	out_flg_busy : BOOL;
	out_flg_Done : BOOL;
	out_var_X : LREAL;
	out_var_Y : LREAL;
	out_var_Z : LREAL;
END_VAR
VAR
	fbi_r_TRIG: R_TRIG;
	var_buf_cavNo: INT;
	var_buf_pocketNo: INT;
	var_xLineNo: INT;
	var_yColmnNo: INT;
	var_foo: INT;
	var_vecP12: LREAL;
	var_vecP13: LREAL;
	var_pitchP13: LREAL;
	var_pitchP12: LREAL;
	var_targetPosX: LREAL;
	var_targetPosY: LREAL;
	var_matrix : ARRAY [1..3, 1..3] OF LREAL;
	var_a: LREAL;
	var_b: LREAL;
	var_c: LREAL;
	var_d: LREAL;
	var_buf_calMode: eP_calculateMode;
	//homography
	var_matrixHomo: ARRAY[0..7] OF ARRAY[0..7] OF LREAL;
	var_originPosX: ARRAY[0..3] OF LREAL;
	var_originPosY: ARRAY[0..3] OF LREAL;
	var_marixPivot: ARRAY[0..7] OF LREAL;
	var_i: INT;
	var_j: INT;
	var_pivot: INT;
	//var_matrixA: ARRAY[0..7] OF ARRAY [0..7] OF LREAL;
	//var_amax: LREAL;
	//var_Tmp: LREAL;
	//var_aryPivot: ARRAY[0..7] OF LREAL;
	//var_j: INT;
	
	var_matrixC: ARRAY[0..7] OF ARRAY[0..7] OF LREAL;
	var_matrixD: ARRAY[0..7] OF ARRAY[0..7] OF LREAL;
	var_hi: INT;
	var_aryA: ARRAY[0..7] OF  LREAL;
	
	
END_VAR

fbi_r_TRIG(CLK:= in_flg_run, Q=> );
out_flg_run := in_flg_run;

IF fbi_r_TRIG.Q THEN
	var_buf_cavNo := in_var_cavNo;
	var_buf_pocketNo := in_var_pocketNo;
	var_buf_calMode := in_var_calculateMode;
	out_flg_busy := TRUE;
END_IF

IF out_flg_Done THEN
	out_flg_busy := FALSE;
END_IF
//caluculate target pocket no
IF out_flg_busy THEN
		IF var_ref_productInfo.bottomPocketQty <> 0 THEN
			var_foo := DINT_TO_INT(TRUNC(var_buf_pocketNo / var_ref_productInfo.bottomPocketQty));
		END_IF
	IF var_foo < 1 THEN
		var_xLineNo := var_buf_pocketNo;
		var_yColmnNo := 1;
	ELSIF var_foo >= 1 THEN
		IF var_foo * var_ref_productInfo.bottomPocketQty = in_var_pocketNo THEN
			var_xLineNo := var_buf_pocketNo - (var_ref_productInfo.bottomPocketQty * (var_foo-1));
			var_yColmnNo := var_foo ;
		ELSE
			var_xLineNo := var_buf_pocketNo - (var_ref_productInfo.bottomPocketQty * var_foo);
			var_yColmnNo := var_foo + 1;
		END_IF
	END_IF

    (*          
    
                      back         
      X - - P[2] ---------------- P[1] 
           /                    /|
          /        tray        / |
         /                    /  Z
        /                    /
       P[4]------------------ P[3]
                           /
                          /
                         Y
	          front
	*)
	

//-----------------------------------------------------------------------------------------------------------------------------
	CASE var_buf_calMode OF
		eP_calculateMode.Affine:
			//length
			var_vecP12 := SQRT(EXPT((var_ref_productInfo.teachPos.palletize.upperLower[gvl_param.var_currentTrayPos].cav[var_buf_cavNo].Pos[2].x - var_ref_productInfo.teachPos.palletize.upperLower[gvl_param.var_currentTrayPos].cav[var_buf_cavNo].Pos[1].x),2) + EXPT((var_ref_productInfo.teachPos.palletize.upperLower[gvl_param.var_currentTrayPos].cav[var_buf_cavNo].Pos[2].y - var_ref_productInfo.teachPos.palletize.upperLower[gvl_param.var_currentTrayPos].cav[var_buf_cavNo].Pos[1].y),2));
			var_vecP13 := SQRT(EXPT((var_ref_productInfo.teachPos.palletize.upperLower[gvl_param.var_currentTrayPos].cav[var_buf_cavNo].Pos[3].x - var_ref_productInfo.teachPos.palletize.upperLower[gvl_param.var_currentTrayPos].cav[var_buf_cavNo].Pos[1].x),2) + EXPT((var_ref_productInfo.teachPos.palletize.upperLower[gvl_param.var_currentTrayPos].cav[var_buf_cavNo].Pos[3].y - var_ref_productInfo.teachPos.palletize.upperLower[gvl_param.var_currentTrayPos].cav[var_buf_cavNo].Pos[1].y),2));
			
			//pitch
			IF var_ref_productInfo.bottomPocketQty = 1 THEN
				var_pitchP12 := var_vecP12;
				var_pitchP13 := var_vecP13 / (var_ref_productInfo.vertivalPocketQty - 1);
			ELSIF var_ref_productInfo.vertivalPocketQty = 1 THEN
				var_pitchP12 := var_vecP12 / (var_ref_productInfo.bottomPocketQty - 1);
				var_pitchP13 := var_vecP13;
			ELSE
				var_pitchP12 := var_vecP12 / (var_ref_productInfo.bottomPocketQty - 1);
				var_pitchP13 := var_vecP13 / (var_ref_productInfo.vertivalPocketQty - 1);
			END_IF
			
			
			//target coordinate data (origin data)
			var_targetPosX := ((var_xLineNo - 1) * var_pitchP12);
			var_targetPosY := ((var_yColmnNo - 1) * var_pitchP13);
			
			//genarate affine transform matrix
			IF var_vecP12 = 0 THEN
				var_matrix[1,1] := 0;
			 	var_matrix[1,2] := -var_ref_productInfo.teachPos.palletize.upperLower[gvl_param.var_currentTrayPos].cav[var_buf_cavNo].Pos[1].x/var_vecP13+var_ref_productInfo.teachPos.palletize.upperLower[gvl_param.var_currentTrayPos].cav[var_buf_cavNo].Pos[3].x/var_vecP13;
			 	var_matrix[1,3] := var_ref_productInfo.teachPos.palletize.upperLower[gvl_param.var_currentTrayPos].cav[var_buf_cavNo].Pos[1].x;
		
			 	var_matrix[2,1] := 0;
			 	var_matrix[2,2] := -var_ref_productInfo.teachPos.palletize.upperLower[gvl_param.var_currentTrayPos].cav[var_buf_cavNo].Pos[1].y/var_vecP13+var_ref_productInfo.teachPos.palletize.upperLower[gvl_param.var_currentTrayPos].cav[var_buf_cavNo].Pos[3].y/var_vecP13;
			 	var_matrix[2,3] := var_ref_productInfo.teachPos.palletize.upperLower[gvl_param.var_currentTrayPos].cav[var_buf_cavNo].Pos[1].y;
			
			  	var_matrix[3,1] := 0;
			  	var_matrix[3,2] := 0;
			  	var_matrix[3,3] := 1;
			ELSIF var_vecP13 = 0 THEN
				var_matrix[1,1] := -var_ref_productInfo.teachPos.palletize.upperLower[gvl_param.var_currentTrayPos].cav[var_buf_cavNo].Pos[1].x/var_vecP12+var_ref_productInfo.teachPos.palletize.upperLower[gvl_param.var_currentTrayPos].cav[var_buf_cavNo].Pos[2].x/var_vecP12;
			 	var_matrix[1,2] := 0;
			 	var_matrix[1,3] := var_ref_productInfo.teachPos.palletize.upperLower[gvl_param.var_currentTrayPos].cav[var_buf_cavNo].Pos[1].x;
		
			 	var_matrix[2,1] := -var_ref_productInfo.teachPos.palletize.upperLower[gvl_param.var_currentTrayPos].cav[var_buf_cavNo].Pos[1].y/var_vecP12+var_ref_productInfo.teachPos.palletize.upperLower[gvl_param.var_currentTrayPos].cav[var_buf_cavNo].Pos[2].y/var_vecP12;
			 	var_matrix[2,2] := 0;
			 	var_matrix[2,3] := var_ref_productInfo.teachPos.palletize.upperLower[gvl_param.var_currentTrayPos].cav[var_buf_cavNo].Pos[1].y;
			
			  	var_matrix[3,1] := 0;
			  	var_matrix[3,2] := 0;
			  	var_matrix[3,3] := 1;
			ELSE
				var_matrix[1,1] := -var_ref_productInfo.teachPos.palletize.upperLower[gvl_param.var_currentTrayPos].cav[var_buf_cavNo].Pos[1].x/var_vecP12+var_ref_productInfo.teachPos.palletize.upperLower[gvl_param.var_currentTrayPos].cav[var_buf_cavNo].Pos[2].x/var_vecP12;
			 	var_matrix[1,2] := -var_ref_productInfo.teachPos.palletize.upperLower[gvl_param.var_currentTrayPos].cav[var_buf_cavNo].Pos[1].x/var_vecP13+var_ref_productInfo.teachPos.palletize.upperLower[gvl_param.var_currentTrayPos].cav[var_buf_cavNo].Pos[3].x/var_vecP13;
			 	var_matrix[1,3] := var_ref_productInfo.teachPos.palletize.upperLower[gvl_param.var_currentTrayPos].cav[var_buf_cavNo].Pos[1].x;
		
			 	var_matrix[2,1] := -var_ref_productInfo.teachPos.palletize.upperLower[gvl_param.var_currentTrayPos].cav[var_buf_cavNo].Pos[1].y/var_vecP12+var_ref_productInfo.teachPos.palletize.upperLower[gvl_param.var_currentTrayPos].cav[var_buf_cavNo].Pos[2].y/var_vecP12;
			 	var_matrix[2,2] := -var_ref_productInfo.teachPos.palletize.upperLower[gvl_param.var_currentTrayPos].cav[var_buf_cavNo].Pos[1].y/var_vecP13+var_ref_productInfo.teachPos.palletize.upperLower[gvl_param.var_currentTrayPos].cav[var_buf_cavNo].Pos[3].y/var_vecP13;
			 	var_matrix[2,3] := var_ref_productInfo.teachPos.palletize.upperLower[gvl_param.var_currentTrayPos].cav[var_buf_cavNo].Pos[1].y;
			
			  	var_matrix[3,1] := 0;
			  	var_matrix[3,2] := 0;
			  	var_matrix[3,3] := 1;
			END_IF

			  
			  
			  //caluculate Axis Z coordinate data
			var_a := (var_ref_productInfo.teachPos.palletize.upperLower[gvl_param.var_currentTrayPos].cav[var_buf_cavNo].Pos[2].y - var_ref_productInfo.teachPos.palletize.upperLower[gvl_param.var_currentTrayPos].cav[var_buf_cavNo].Pos[1].y) * (var_ref_productInfo.teachPos.palletize.upperLower[gvl_param.var_currentTrayPos].cav[var_buf_cavNo].Pos[3].z - var_ref_productInfo.teachPos.palletize.upperLower[gvl_param.var_currentTrayPos].cav[var_buf_cavNo].Pos[1].z) - (var_ref_productInfo.teachPos.palletize.upperLower[gvl_param.var_currentTrayPos].cav[var_buf_cavNo].Pos[3].y - var_ref_productInfo.teachPos.palletize.upperLower[gvl_param.var_currentTrayPos].cav[var_buf_cavNo].Pos[1].y) * (var_ref_productInfo.teachPos.palletize.upperLower[gvl_param.var_currentTrayPos].cav[var_buf_cavNo].Pos[2].z - var_ref_productInfo.teachPos.palletize.upperLower[gvl_param.var_currentTrayPos].cav[var_buf_cavNo].Pos[1].z);
			var_b := (var_ref_productInfo.teachPos.palletize.upperLower[gvl_param.var_currentTrayPos].cav[var_buf_cavNo].Pos[2].z - var_ref_productInfo.teachPos.palletize.upperLower[gvl_param.var_currentTrayPos].cav[var_buf_cavNo].Pos[1].z) * (var_ref_productInfo.teachPos.palletize.upperLower[gvl_param.var_currentTrayPos].cav[var_buf_cavNo].Pos[3].x - var_ref_productInfo.teachPos.palletize.upperLower[gvl_param.var_currentTrayPos].cav[var_buf_cavNo].Pos[1].x) - (var_ref_productInfo.teachPos.palletize.upperLower[gvl_param.var_currentTrayPos].cav[var_buf_cavNo].Pos[3].z - var_ref_productInfo.teachPos.palletize.upperLower[gvl_param.var_currentTrayPos].cav[var_buf_cavNo].Pos[1].z) * (var_ref_productInfo.teachPos.palletize.upperLower[gvl_param.var_currentTrayPos].cav[var_buf_cavNo].Pos[2].x - var_ref_productInfo.teachPos.palletize.upperLower[gvl_param.var_currentTrayPos].cav[var_buf_cavNo].Pos[1].x);
			var_c := (var_ref_productInfo.teachPos.palletize.upperLower[gvl_param.var_currentTrayPos].cav[var_buf_cavNo].Pos[2].x - var_ref_productInfo.teachPos.palletize.upperLower[gvl_param.var_currentTrayPos].cav[var_buf_cavNo].Pos[1].x) * (var_ref_productInfo.teachPos.palletize.upperLower[gvl_param.var_currentTrayPos].cav[var_buf_cavNo].Pos[3].y - var_ref_productInfo.teachPos.palletize.upperLower[gvl_param.var_currentTrayPos].cav[var_buf_cavNo].Pos[1].y) - (var_ref_productInfo.teachPos.palletize.upperLower[gvl_param.var_currentTrayPos].cav[var_buf_cavNo].Pos[3].x - var_ref_productInfo.teachPos.palletize.upperLower[gvl_param.var_currentTrayPos].cav[var_buf_cavNo].Pos[1].x) * (var_ref_productInfo.teachPos.palletize.upperLower[gvl_param.var_currentTrayPos].cav[var_buf_cavNo].Pos[2].y - var_ref_productInfo.teachPos.palletize.upperLower[gvl_param.var_currentTrayPos].cav[var_buf_cavNo].Pos[1].y);
			var_d := -((var_a * var_ref_productInfo.teachPos.palletize.upperLower[gvl_param.var_currentTrayPos].cav[var_buf_cavNo].Pos[1].x) + (var_b * var_ref_productInfo.teachPos.palletize.upperLower[gvl_param.var_currentTrayPos].cav[var_buf_cavNo].Pos[1].y) + (var_c * var_ref_productInfo.teachPos.palletize.upperLower[gvl_param.var_currentTrayPos].cav[var_buf_cavNo].Pos[1].z));
			
			// caluculate (afiine transform matrix * target coordinate data)
			out_var_X := (var_matrix[1,1] * var_targetPosX) + (var_matrix[1,2] * var_targetPosY) + var_matrix[1,3];
			out_var_Y := (var_matrix[2,1] * var_targetPosX) + (var_matrix[2,2] * var_targetPosY) + var_matrix[2,3];
			IF var_c <> 0 THEN
				out_var_Z := -((var_a * out_var_X) + (var_b * out_var_Y) + var_d) / var_c;
			ELSE
				out_var_Z := var_ref_productInfo.teachPos.palletize.upperLower[gvl_param.var_currentTrayPos].cav[var_buf_cavNo].Pos[1].z;
			END_IF	
			out_flg_Done := TRUE;
		eP_calculateMode.Homography:
			//
			out_flg_Done := FALSE;
	END_CASE

ELSE
	out_flg_Done := FALSE;
	
END_IF

END_FUNCTION_BLOCK

// ---- FBs/fb_operationElecylinder.TcPOU
FUNCTION_BLOCK fb_operationElecylinder
VAR_INPUT
END_VAR
VAR_OUTPUT
END_VAR
VAR
	SFCInit: bool;
	TranPosDone: BOOL;
	TranNegDone: BOOL;
	SamplePosDone: BOOL;
	SampleNegDone: BOOL;
	TrayChangePosDone: BOOL;
	TrayChangeNegDone: BOOL;
	flgInitDone: BOOL;
	trn_RotaryNegDone: BOOL;
	trn_RotaryPosDone: BOOL;
	trn_flgInitDone: BOOL;
	var_process: INT;
END_VAR

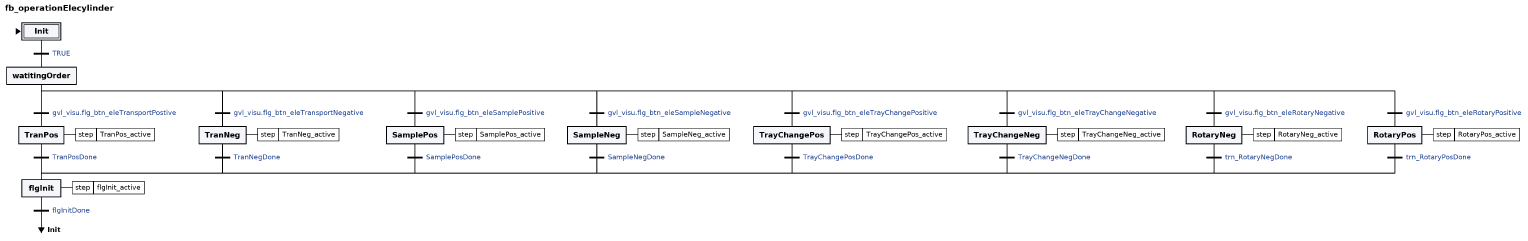
INITIAL_STEP Init:
END_STEP
TRANSITION FROM Init TO watitingOrder
    := TRUE;
END_TRANSITION
STEP watitingOrder:
END_STEP
TRANSITION FROM watitingOrder TO TranPos
    := gvl_visu.flg_btn_eleTransportPostive;
END_TRANSITION
STEP TranPos:
    TranPos_active(N);  // step action
END_STEP
TRANSITION FROM TranPos TO flgInit
    := TranPosDone;
END_TRANSITION
TRANSITION FROM watitingOrder TO TranNeg
    := gvl_visu.flg_btn_eleTransportNegative;
END_TRANSITION
STEP TranNeg:
    TranNeg_active(N);  // step action
END_STEP
TRANSITION FROM TranNeg TO flgInit
    := TranNegDone;
END_TRANSITION
TRANSITION FROM watitingOrder TO SamplePos
    := gvl_visu.flg_btn_eleSamplePositive;
END_TRANSITION
STEP SamplePos:
    SamplePos_active(N);  // step action
END_STEP
TRANSITION FROM SamplePos TO flgInit
    := SamplePosDone;
END_TRANSITION
TRANSITION FROM watitingOrder TO SampleNeg
    := gvl_visu.flg_btn_eleSampleNegative;
END_TRANSITION
STEP SampleNeg:
    SampleNeg_active(N);  // step action
END_STEP
TRANSITION FROM SampleNeg TO flgInit
    := SampleNegDone;
END_TRANSITION
TRANSITION FROM watitingOrder TO TrayChangePos
    := gvl_visu.flg_btn_eleTrayChangePositive;
END_TRANSITION
STEP TrayChangePos:
    TrayChangePos_active(N);  // step action
END_STEP
TRANSITION FROM TrayChangePos TO flgInit
    := TrayChangePosDone;
END_TRANSITION
TRANSITION FROM watitingOrder TO TrayChangeNeg
    := gvl_visu.flg_btn_eleTrayChangeNegative;
END_TRANSITION
STEP TrayChangeNeg:
    TrayChangeNeg_active(N);  // step action
END_STEP
TRANSITION FROM TrayChangeNeg TO flgInit
    := TrayChangeNegDone;
END_TRANSITION
TRANSITION FROM watitingOrder TO RotaryNeg
    := gvl_visu.flg_btn_eleRotaryNegative;
END_TRANSITION
STEP RotaryNeg:
    RotaryNeg_active(N);  // step action
END_STEP
TRANSITION FROM RotaryNeg TO flgInit
    := trn_RotaryNegDone;
END_TRANSITION
TRANSITION FROM watitingOrder TO RotaryPos
    := gvl_visu.flg_btn_eleRotaryPositive;
END_TRANSITION
STEP RotaryPos:
    RotaryPos_active(N);  // step action
END_STEP
TRANSITION FROM RotaryPos TO flgInit
    := trn_RotaryPosDone;
END_TRANSITION
STEP flgInit:
    flgInit_active(N);  // step action
END_STEP
TRANSITION FROM flgInit TO Init
    := flgInitDone;
END_TRANSITION

ACTION flgInit_active:
IF flgInit._x AND flgInit.x = FALSE THEN
	flgInitDone:= FALSE;
	gvl_visu.flg_btn_eleTransportPostive := FALSE;
	gvl_visu.flg_btn_eleTransportNegative := FALSE;
	gvl_visu.flg_btn_eleSamplePositive := FALSE;
	gvl_visu.flg_btn_eleSampleNegative := FALSE;
	gvl_visu.flg_btn_eleTrayChangePositive := FALSE;
	gvl_visu.flg_btn_eleTrayChangeNegative := FALSE;
	gvl_visu.flg_btn_eleRotaryPositive := FALSE;
	gvl_visu.flg_btn_eleRotaryNegative := FALSE;
ELSIF flgInit._x AND flgInit.x THEN
	flgInitDone := TRUE;
END_IF
END_ACTION

PROPERTY p_Init : bool
GET
p_init := THIS^.SFCInit;
END_GET
SET
THIS^.SFCInit := p_init;
END_SET
END_PROPERTY

ACTION RotaryNeg_active:
IF RotaryNeg._x AND RotaryNeg.x = FALSE THEN
	trn_RotaryNegDone := FALSE;
	gvl_elecylinder.fbi_axisRotary.in_flg_run := FALSE;
	gvl_elecylinder.fbi_axisRotary.in_var_moveMode := eP_eleMoveMode.eleA;
	var_process := 0;
ELSIF RotaryNeg._x AND RotaryNeg.x THEN
	CASE var_process OF
		0:
			gvl_elecylinder.fbi_axisRotary.in_flg_run := TRUE;
			var_process := 1;
		1:
			IF gvl_elecylinder.fbi_axisRotary.out_flg_Done THEN
				gvl_elecylinder.fbi_axisRotary.in_flg_run := FALSE;
				trn_RotaryNegDone := TRUE;
			END_IF
	END_CASE
END_IF
END_ACTION

ACTION RotaryPos_active:
IF RotaryPos._x AND RotaryPos.x = FALSE THEN
	trn_RotaryPosDone := FALSE;
	gvl_elecylinder.fbi_axisRotary.in_flg_run := FALSE;
	gvl_elecylinder.fbi_axisRotary.in_var_moveMode := eP_eleMoveMode.eleB;
	var_process := 0;
ELSIF RotaryPos._x AND RotaryPos.x THEN
	CASE var_process OF
		0:
			gvl_elecylinder.fbi_axisRotary.in_flg_run := TRUE;
			var_process :=1;
		1:
			IF gvl_elecylinder.fbi_axisRotary.out_flg_Done THEN
				gvl_elecylinder.fbi_axisRotary.in_flg_run := FALSE;
				trn_RotaryPosDone := TRUE;
			END_IF
	END_CASE
END_IF
END_ACTION

ACTION SampleNeg_active:
IF SampleNeg._x AND SampleNeg.x = FALSE THEN
	SampleNegDone := FALSE;
	gvl_elecylinder.fbi_axisSample.in_flg_run := FALSE;
	gvl_elecylinder.fbi_axisSample.in_var_moveMode := eP_eleMoveMode.eleA;
	var_process := 0;
ELSIF SampleNeg._x AND SampleNeg.x THEN
	CASE var_process OF
		0:
			gvl_elecylinder.fbi_axisSample.in_flg_run := TRUE;
			var_process := 1;
		1:
			IF gvl_elecylinder.fbi_axisSample.out_flg_Done THEN
				gvl_elecylinder.fbi_axisSample.in_flg_run := FALSE;
				SampleNegDone := TRUE;
			END_IF
	END_CASE
END_IF
END_ACTION

ACTION SamplePos_active:
IF SamplePos._x AND SamplePos.x = FALSE THEN
	SamplePosDone := FALSE;
	gvl_elecylinder.fbi_axisSample.in_flg_run := FALSE;
	gvl_elecylinder.fbi_axisSample.in_var_moveMode := eP_eleMoveMode.eleB;
	var_process := 0;
ELSIF SamplePos._x AND SamplePos.x THEN
	CASE var_process OF
		0:
			gvl_elecylinder.fbi_axisSample.in_flg_run := TRUE;
			var_process := 1;
		1:
			IF gvl_elecylinder.fbi_axisSample.out_flg_Done THEN
				gvl_elecylinder.fbi_axisSample.in_flg_run := FALSE;
				SamplePosDone := TRUE;
			END_IF
	END_CASE
END_IF
END_ACTION

ACTION TranNeg_active:
IF TranNeg._x AND TranNeg.x = FALSE THEN
	TranNegDone := FALSE;
	gvl_elecylinder.fbi_axisTransport.in_flg_run := FALSE;
	gvl_elecylinder.fbi_axisTransport.in_var_moveMode := eP_eleMoveMode.eleA;
	var_process := 0;
ELSIF TranNeg._x AND TranNeg.x THEN
	CASE var_process OF
		0:
			gvl_elecylinder.fbi_axisTransport.in_flg_run := TRUE;
			var_process := 1;
		1:
			IF gvl_elecylinder.fbi_axisTransport.out_flg_Done THEN
				gvl_elecylinder.fbi_axisTransport.in_flg_run := FALSE;
				TranNegDone := TRUE;
			END_IF
	END_CASE
END_IF
END_ACTION

ACTION TranPos_active:
IF TranPos._x AND TranPos.x = FALSE THEN
	TranPosDone := FALSE;
	gvl_elecylinder.fbi_axisTransport.in_flg_run := FALSE;
	gvl_elecylinder.fbi_axisTransport.in_var_moveMode := eP_eleMoveMode.eleB;
	var_process := 0;
ELSIF TranPos._x AND TranPos.x THEN
	CASE var_process OF
		0:
			gvl_elecylinder.fbi_axisTransport.in_flg_run := TRUE;
			var_process := 1;
		1:
			IF gvl_elecylinder.fbi_axisTransport.out_flg_Done THEN
				TranPosDone := TRUE;
			END_IF
	END_CASE
END_IF
END_ACTION

ACTION TrayChangeNeg_active:
IF TrayChangeNeg._x AND TrayChangeNeg.x = FALSE THEN
	TrayChangeNegDone := FALSE;
	gvl_elecylinder.fbi_axisTrayChange.in_flg_run := FALSE;
	gvl_elecylinder.fbi_axisTrayChange.in_var_moveMode := eP_eleMoveMode.eleA;
	var_process := 0;
ELSIF TrayChangeNeg._x AND TrayChangeNeg.x THEN
	CASE var_process OF
		0:
			gvl_axis.ref_z.Position := 50;
			gvl_axis.ref_z.Execute := TRUE;
			var_process := 1;
		1:
			IF gvl_axis.ref_z.Done THEN
				gvl_axis.ref_z.Execute := FALSE;
				var_process := 2;
			END_IF
		2:
			gvl_elecylinder.fbi_axisTrayChange.in_flg_run := TRUE;
			var_process := 3;
		3:
			IF gvl_elecylinder.fbi_axisTrayChange.out_flg_Done THEN
				gvl_elecylinder.fbi_axisTrayChange.in_flg_run := FALSE;
				TrayChangeNegDone := TRUE;
			END_IF
	END_CASE
END_IF
END_ACTION

ACTION TrayChangePos_active:
IF TrayChangePos._x AND TrayChangePos.x = FALSE THEN
	TrayChangePosDone := FALSE;
	gvl_elecylinder.fbi_axisTrayChange.in_flg_run := FALSE;
	gvl_elecylinder.fbi_axisTrayChange.in_var_moveMode := eP_eleMoveMode.eleB;
	var_process := 0;
ELSIF TrayChangePos._x AND TrayChangePos.x THEN
	CASE var_process OF
		0:
			gvl_axis.ref_z.Position := 50;
			gvl_axis.ref_z.Execute := TRUE;
			var_process := 1;
		1:
			IF gvl_axis.ref_z.Done THEN
				gvl_axis.ref_z.Execute := FALSE;
				var_process := 2;
			END_IF
		2:
			gvl_elecylinder.fbi_axisTrayChange.in_flg_run := TRUE;
			var_process := 3;
		3:
			IF gvl_elecylinder.fbi_axisTrayChange.out_flg_Done THEN
				gvl_elecylinder.fbi_axisTrayChange.in_flg_run := FALSE;
				TrayChangePosDone := TRUE;
			END_IF
	END_CASE
END_IF
END_ACTION

END_FUNCTION_BLOCK

// ---- FBs/gateMeasurementModule/fb_gm_operationElecylinder.TcPOU
FUNCTION_BLOCK fb_gm_operationElecylinder
VAR_INPUT
END_VAR
VAR_OUTPUT
END_VAR
VAR
	SFCInit: bool;
	TranPosDone: BOOL;
	TranNegDone: BOOL;
	flgInitDone: BOOL;
	PickUpPosDone: BOOL;
	PickUpNegDone: BOOL;
	var_process: INT;
END_VAR

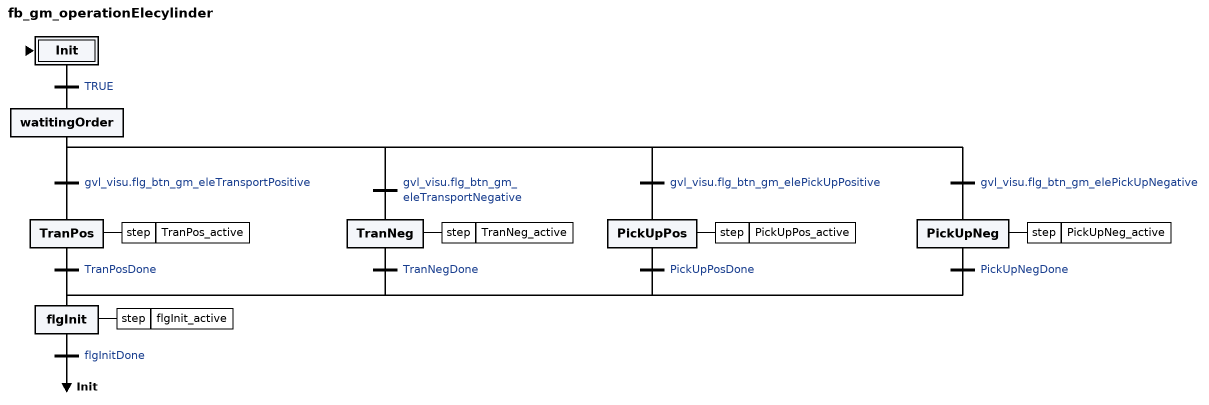
INITIAL_STEP Init:
END_STEP
TRANSITION FROM Init TO watitingOrder
    := TRUE;
END_TRANSITION
STEP watitingOrder:
END_STEP
TRANSITION FROM watitingOrder TO TranPos
    := gvl_visu.flg_btn_gm_eleTransportPositive;
END_TRANSITION
STEP TranPos:
    TranPos_active(N);  // step action
END_STEP
TRANSITION FROM TranPos TO flgInit
    := TranPosDone;
END_TRANSITION
TRANSITION FROM watitingOrder TO TranNeg
    := gvl_visu.flg_btn_gm_eleTransportNegative;
END_TRANSITION
STEP TranNeg:
    TranNeg_active(N);  // step action
END_STEP
TRANSITION FROM TranNeg TO flgInit
    := TranNegDone;
END_TRANSITION
TRANSITION FROM watitingOrder TO PickUpPos
    := gvl_visu.flg_btn_gm_elePickUpPositive;
END_TRANSITION
STEP PickUpPos:
    PickUpPos_active(N);  // step action
END_STEP
TRANSITION FROM PickUpPos TO flgInit
    := PickUpPosDone;
END_TRANSITION
TRANSITION FROM watitingOrder TO PickUpNeg
    := gvl_visu.flg_btn_gm_elePickUpNegative;
END_TRANSITION
STEP PickUpNeg:
    PickUpNeg_active(N);  // step action
END_STEP
TRANSITION FROM PickUpNeg TO flgInit
    := PickUpNegDone;
END_TRANSITION
STEP flgInit:
    flgInit_active(N);  // step action
END_STEP
TRANSITION FROM flgInit TO Init
    := flgInitDone;
END_TRANSITION

ACTION flgInit_active:
IF flgInit._x AND flgInit.x = FALSE THEN
	flgInitDone:= FALSE;
	gvl_visu.flg_btn_gm_eleTransportPositive := FALSE;
	gvl_visu.flg_btn_gm_eleTransportNegative := FALSE;
	gvl_visu.flg_btn_gm_elePickUpPositive := FALSE;
	gvl_visu.flg_btn_gm_elePickUpNegative := FALSE;
	gvl_visu.flg_btn_eleSamplePositive := FALSE;
	gvl_visu.flg_btn_eleSampleNegative := FALSE;
	gvl_visu.flg_btn_eleTrayChangePositive := FALSE;
	gvl_visu.flg_btn_eleTrayChangeNegative := FALSE;
	gvl_visu.flg_btn_eleRotaryPositive := FALSE;
	gvl_visu.flg_btn_eleRotaryNegative := FALSE;
ELSIF flgInit._x AND flgInit.x THEN
	flgInitDone := TRUE;
END_IF
END_ACTION

PROPERTY p_Init : bool
GET
p_init := THIS^.SFCInit;
END_GET
SET
THIS^.SFCInit := p_init;
END_SET
END_PROPERTY

ACTION PickUpNeg_active:
IF PickUpNeg._x AND PickUpNeg.x = FALSE THEN
	PickUpNegDone := FALSE;
	gvl_elecylinder.fbi_gm_axisPickUp.in_flg_run := FALSE;
	gvl_elecylinder.fbi_gm_axisPickUp.in_var_moveMode := eP_eleMoveMode.eleA;
	var_process := 0;
ELSIF PickUpNeg._x AND PickUpNeg.x THEN
	CASE var_process OF
		0:
			gvl_elecylinder.fbi_gm_axisPickUp.in_flg_run := TRUE;
			var_process := 1;
		1:
			IF gvl_elecylinder.fbi_gm_axisPickUp.out_flg_Done THEN
				gvl_elecylinder.fbi_gm_axisPickUp.in_flg_run := FALSE;
				PickUpNegDone := TRUE;
			END_IF
	END_CASE
END_IF
END_ACTION

ACTION PickUpPos_active:
IF PickUpPos._x AND PickUpPos.x = FALSE THEN
	PickUpPosDone := FALSE;
	gvl_elecylinder.fbi_gm_axisPickUp.in_flg_run := FALSE;
	gvl_elecylinder.fbi_gm_axisPickUp.in_var_moveMode := eP_eleMoveMode.eleB;
	var_process := 0;
ELSIF PickUpPos._x AND PickUpPos.x THEN
	CASE var_process OF
		0:
			gvl_elecylinder.fbi_gm_axisPickUp.in_flg_run := TRUE;
			var_process := 1;
		1:
			IF gvl_elecylinder.fbi_gm_axisPickUp.out_flg_Done THEN
				gvl_elecylinder.fbi_gm_axisPickUp.in_flg_run := FALSE;
				PickUpPosDone := TRUE;
			END_IF
	END_CASE
END_IF
END_ACTION

ACTION TranNeg_active:
IF TranNeg._x AND TranNeg.x = FALSE THEN
	TranNegDone := FALSE;
	gvl_elecylinder.fbi_gm_axisTransport.in_flg_run := FALSE;
	gvl_elecylinder.fbi_gm_axisTransport.in_var_moveMode := eP_eleMoveMode.eleA;
	var_process := 0;
ELSIF TranNeg._x AND TranNeg.x THEN
	CASE var_process OF
		0:
			gvl_elecylinder.fbi_gm_axisTransport.in_flg_run := TRUE;
			var_process := 1;
		1:
			IF gvl_elecylinder.fbi_gm_axisTransport.out_flg_Done THEN
				gvl_elecylinder.fbi_gm_axisTransport.in_flg_run := FALSE;
				TranNegDone := TRUE;
			END_IF
	END_CASE
END_IF
END_ACTION

ACTION TranPos_active:
IF TranPos._x AND TranPos.x = FALSE THEN
	TranPosDone := FALSE;
	gvl_elecylinder.fbi_gm_axisTransport.in_flg_run := FALSE;
	gvl_elecylinder.fbi_gm_axisTransport.in_var_moveMode := eP_eleMoveMode.eleB;
	var_process := 0;
ELSIF TranPos._x AND TranPos.x THEN
	CASE var_process OF
		0:
			gvl_elecylinder.fbi_gm_axisTransport.in_flg_run := TRUE;
			var_process := 1;
		1:
			IF gvl_elecylinder.fbi_gm_axisTransport.out_flg_Done THEN
				gvl_elecylinder.fbi_gm_axisTransport.in_flg_run := FALSE;
				TranPosDone := TRUE;
			END_IF
	END_CASE
END_IF
END_ACTION

END_FUNCTION_BLOCK

// ---- FBs/fb_oeprationChuck.TcPOU
FUNCTION_BLOCK fb_oeprationChuck
VAR_INPUT
END_VAR
VAR_OUTPUT
END_VAR
VAR
	SFCInit : bool;
	flgInitDone: BOOL;
	trn_chuckCloseDone: BOOL;
	trn_chuckOpenDone: BOOL;
END_VAR

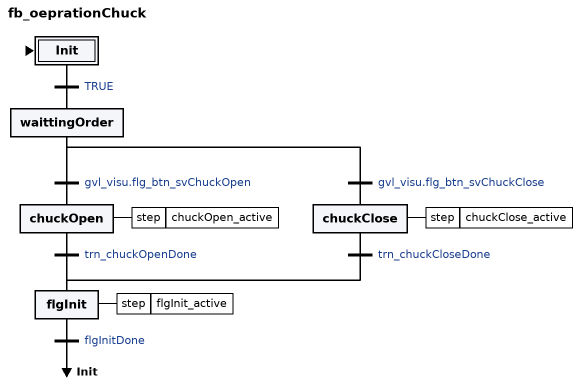
INITIAL_STEP Init:
END_STEP
TRANSITION FROM Init TO waittingOrder
    := TRUE;
END_TRANSITION
STEP waittingOrder:
END_STEP
TRANSITION FROM waittingOrder TO chuckOpen
    := gvl_visu.flg_btn_svChuckOpen;
END_TRANSITION
STEP chuckOpen:
    chuckOpen_active(N);  // step action
END_STEP
TRANSITION FROM chuckOpen TO flgInit
    := trn_chuckOpenDone;
END_TRANSITION
TRANSITION FROM waittingOrder TO chuckClose
    := gvl_visu.flg_btn_svChuckClose;
END_TRANSITION
STEP chuckClose:
    chuckClose_active(N);  // step action
END_STEP
TRANSITION FROM chuckClose TO flgInit
    := trn_chuckCloseDone;
END_TRANSITION
STEP flgInit:
    flgInit_active(N);  // step action
END_STEP
TRANSITION FROM flgInit TO Init
    := flgInitDone;
END_TRANSITION

ACTION chuckClose_active:
IF chuckClose._x AND chuckClose.x = FALSE THEN
	trn_chuckCloseDone := FALSE;
	gvl_solv.fbi_chuck.in_flg_run := FALSE;
	gvl_solv.fbi_chuck.in_var_moveMode := eP_svMoveMode.svB;
ELSIF chuckClose._x AND chuckClose.x THEN
	gvl_solv.fbi_chuck.in_flg_run := TRUE;
	IF gvl_solv.fbi_chuck.out_flg_Done THEN
		gvl_solv.fbi_chuck.in_flg_run := FALSE;
		trn_chuckCloseDone := TRUE;
	END_IF
END_IF
END_ACTION

ACTION chuckOpen_active:
IF chuckOpen._x AND chuckOpen.x = FALSE THEN
	trn_chuckOpenDone := FALSE;
	gvl_solv.fbi_chuck.in_flg_run := FALSE;
	gvl_solv.fbi_chuck.in_var_moveMode := eP_svMoveMode.svA;
ELSIF chuckOpen._x AND chuckOpen.x THEN
	gvl_solv.fbi_chuck.in_flg_run := TRUE;
	IF gvl_solv.fbi_chuck.out_flg_Done THEN
		gvl_solv.fbi_chuck.in_flg_run := FALSE;
		trn_chuckOpenDone := TRUE;
	END_IF
END_IF
END_ACTION

ACTION flgInit_active:
IF flgInit._x AND flgInit.x = FALSE THEN
	flgInitDone := FALSE;
	gvl_visu.flg_btn_svChuckOpen := FALSE;
	gvl_visu.flg_btn_svChuckClose := FALSE;
ELSIF flgInit._x AND flgInit.x THEN
	flgInitDone := TRUE;
END_IF
END_ACTION

PROPERTY p_Init : bool
GET
p_init := THIS^.SFCInit;
END_GET
SET
THIS^.SFCInit := p_Init;
END_SET
END_PROPERTY

END_FUNCTION_BLOCK

// ---- FBs/fb_oeprationPush.TcPOU
FUNCTION_BLOCK fb_oeprationPush
VAR_INPUT
END_VAR
VAR_OUTPUT
END_VAR
VAR
	SFCInit : bool;
	flgInitDone: BOOL;
	trn_chuckOpenDone: BOOL;
	trn_chuckCloseDone: BOOL;
	trn_gm_chuckOpenDone: BOOL;
	trn_gm_chuckCloseDone: BOOL;
END_VAR

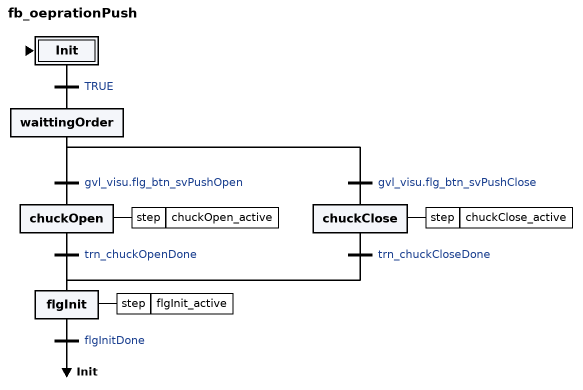
INITIAL_STEP Init:
END_STEP
TRANSITION FROM Init TO waittingOrder
    := TRUE;
END_TRANSITION
STEP waittingOrder:
END_STEP
TRANSITION FROM waittingOrder TO chuckOpen
    := gvl_visu.flg_btn_svPushOpen;
END_TRANSITION
STEP chuckOpen:
    chuckOpen_active(N);  // step action
END_STEP
TRANSITION FROM chuckOpen TO flgInit
    := trn_chuckOpenDone;
END_TRANSITION
TRANSITION FROM waittingOrder TO chuckClose
    := gvl_visu.flg_btn_svPushClose;
END_TRANSITION
STEP chuckClose:
    chuckClose_active(N);  // step action
END_STEP
TRANSITION FROM chuckClose TO flgInit
    := trn_chuckCloseDone;
END_TRANSITION
STEP flgInit:
    flgInit_active(N);  // step action
END_STEP
TRANSITION FROM flgInit TO Init
    := flgInitDone;
END_TRANSITION

ACTION chuckClose_active:
IF chuckClose._x AND chuckClose.x = FALSE THEN
	trn_chuckCloseDone := FALSE;
	gvl_solv.fbi_push.in_flg_run := FALSE;
	gvl_solv.fbi_push.in_var_moveMode := eP_svMoveMode.svB;
ELSIF chuckClose._x AND chuckClose.x THEN
	gvl_solv.fbi_push.in_flg_run := TRUE;
	IF gvl_solv.fbi_push.out_flg_Done THEN
		gvl_solv.fbi_push.in_flg_run := FALSE;
		trn_chuckCloseDone := TRUE;
	END_IF
END_IF
END_ACTION

ACTION chuckOpen_active:
IF chuckOpen._x AND chuckOpen.x = FALSE THEN
	trn_chuckOpenDone := FALSE;
	gvl_solv.fbi_push.in_flg_run := FALSE;
	gvl_solv.fbi_push.in_var_moveMode := eP_svMoveMode.svA;
ELSIF chuckOpen._x AND chuckOpen.x THEN
	gvl_solv.fbi_push.in_flg_run := TRUE;
	IF gvl_solv.fbi_push.out_flg_Done THEN
 		gvl_solv.fbi_push.in_flg_run := FALSE;
		trn_chuckOpenDone := TRUE;
	END_IF
END_IF
END_ACTION

ACTION flgInit_active:
IF flgInit._x AND flgInit.x = FALSE THEN
	flgInitDone := FALSE;
	gvl_visu.flg_btn_svPushOpen := FALSE;
	gvl_visu.flg_btn_svPushClose := FALSE;
ELSIF flgInit._x AND flgInit.x THEN
	flgInitDone := TRUE;
END_IF
END_ACTION

PROPERTY p_Init : bool
GET
p_init := THIS^.SFCInit;
END_GET
SET
THIS^.SFCInit := p_Init;
END_SET
END_PROPERTY

END_FUNCTION_BLOCK

// ---- FBs/fb_operationEjector.TcPOU
FUNCTION_BLOCK fb_operationEjector
VAR_INPUT
END_VAR
VAR_OUTPUT
END_VAR
VAR
	SFCInit : bool;
	flgInitDone: BOOL;
	trn_vacuumOnDone: BOOL;
	trn_vacuumOffDone: BOOL;
	trn_breakOnDone: BOOL;
	trn_breakOffDone: BOOL;
	var_process: INT;
END_VAR

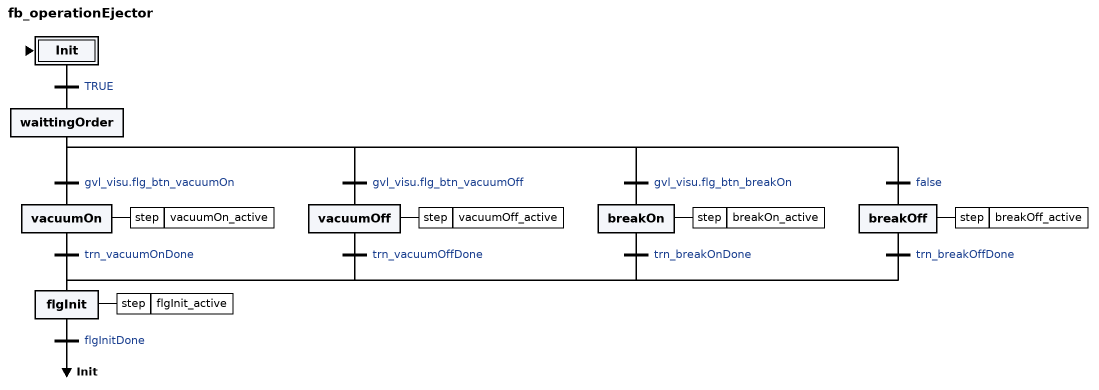
INITIAL_STEP Init:
END_STEP
TRANSITION FROM Init TO waittingOrder
    := TRUE;
END_TRANSITION
STEP waittingOrder:
END_STEP
TRANSITION FROM waittingOrder TO vacuumOn
    := gvl_visu.flg_btn_vacuumOn;
END_TRANSITION
STEP vacuumOn:
    vacuumOn_active(N);  // step action
END_STEP
TRANSITION FROM vacuumOn TO flgInit
    := trn_vacuumOnDone;
END_TRANSITION
TRANSITION FROM waittingOrder TO vacuumOff
    := gvl_visu.flg_btn_vacuumOff;
END_TRANSITION
STEP vacuumOff:
    vacuumOff_active(N);  // step action
END_STEP
TRANSITION FROM vacuumOff TO flgInit
    := trn_vacuumOffDone;
END_TRANSITION
TRANSITION FROM waittingOrder TO breakOn
    := gvl_visu.flg_btn_breakOn;
END_TRANSITION
STEP breakOn:
    breakOn_active(N);  // step action
END_STEP
TRANSITION FROM breakOn TO flgInit
    := trn_breakOnDone;
END_TRANSITION
TRANSITION FROM waittingOrder TO breakOff
    := false;
END_TRANSITION
STEP breakOff:
    breakOff_active(N);  // step action
END_STEP
TRANSITION FROM breakOff TO flgInit
    := trn_breakOffDone;
END_TRANSITION
STEP flgInit:
    flgInit_active(N);  // step action
END_STEP
TRANSITION FROM flgInit TO Init
    := flgInitDone;
END_TRANSITION

ACTION breakOff_active:
IF breakOff._x AND breakOff.x = FALSE THEN
	trn_breakOffDone := FALSE;
	gvl_solv.fbi_ejector.in_flg_run := FALSE;
	gvl_solv.fbi_ejector.in_var_vacMode := eP_ejevacMode.breakOff;
	var_process := 0;
ELSIF breakOff._x AND breakOff.x THEN
	CASE var_process OF
		0:
			gvl_solv.fbi_ejector.in_flg_run := TRUE;
			var_process := 1;
		1:
			IF gvl_solv.fbi_ejector.out_flg_Done THEN
				gvl_solv.fbi_ejector.in_flg_run := FALSE;
				trn_breakOffDone := TRUE;
			END_IF
	END_CASE
END_IF
END_ACTION

ACTION breakOn_active:
IF breakOn._x AND breakOn.x = FALSE THEN
	trn_breakOnDone := FALSE;
	gvl_solv.fbi_ejector.in_flg_run := FALSE;
	gvl_solv.fbi_ejector.in_var_vacMode := eP_ejevacMode.break;
	var_process := 0;
ELSIF breakOn._x AND breakOn._x THEN
	CASE var_process OF
		0:
			gvl_solv.fbi_ejector.in_flg_run := TRUE;
			var_process := 1;
		1:
			IF gvl_solv.fbi_ejector.out_flg_Done THEN
				gvl_solv.fbi_ejector.in_flg_run := FALSE;
				trn_breakOnDone := TRUE;
			END_IF
	END_CASE
END_IF
END_ACTION

ACTION flgInit_active:
IF flgInit._x AND flgInit.x = FALSE THEN
	flgInitDone := FALSE;
	gvl_visu.flg_btn_vacuumOn := FALSE;
	gvl_visu.flg_btn_vacuumOff := FALSE;
	gvl_visu.flg_btn_breakOn := FALSE;
	
ELSIF flgInit._x AND flgInit.x THEN
	flgInitDone := TRUE;
END_IF
END_ACTION

PROPERTY p_Init : bool
GET
p_init := THIS^.SFCInit;
END_GET
SET
THIS^.SFCInit := p_Init;
END_SET
END_PROPERTY

ACTION vacuumOff_active:
IF vacuumOff._x AND vacuumOff.x = FALSE THEN
	trn_vacuumOffDone := FALSE;
	gvl_solv.fbi_ejector.in_flg_run := FALSE;
	gvl_solv.fbi_ejector.in_var_vacMode := eP_ejevacMode.vacOff;
	var_process := 0;
ELSIF vacuumOff._x AND vacuumOff.x THEN
	CASE var_process OF
		0:
			gvl_solv.fbi_ejector.in_flg_run := TRUE;
			var_process :=1;
		1:
			IF gvl_solv.fbi_ejector.out_flg_Done THEN
				gvl_solv.fbi_ejector.in_flg_run := FALSE;
				trn_vacuumOffDone := TRUE;
			END_IF
	END_CASE
END_IF
END_ACTION

ACTION vacuumOn_active:
IF vacuumOn._x AND vacuumOn.x = FALSE THEN
	trn_vacuumOnDone := FALSE;
	gvl_solv.fbi_ejector.in_flg_run := FALSE;
	gvl_solv.fbi_ejector.in_var_vacMode := eP_ejevacMode.halt;
	var_process := 0;
ELSIF vacuumOn._x AND vacuumOn.x THEN
	CASE var_process OF
		0:
			gvl_solv.fbi_ejector.in_flg_run := TRUE;
			var_process := 1;
		1:
			IF gvl_solv.fbi_ejector.out_flg_Done THEN
				gvl_solv.fbi_ejector.in_flg_run := FALSE;
				trn_vacuumOnDone := TRUE;
			END_IF
	END_CASE
END_IF
END_ACTION

END_FUNCTION_BLOCK

// ---- FBs/gateMeasurementModule/fb_gm_operationEjector.TcPOU
FUNCTION_BLOCK fb_gm_operationEjector
VAR_INPUT
END_VAR
VAR_OUTPUT
END_VAR
VAR
	SFCInit : bool;
	flgInitDone: BOOL;
	trn_vacuumOnDone: BOOL;
	trn_vacuumOffDone: BOOL;
	trn_breakOnDone: BOOL;
	trn_breakOffDone: BOOL;
	var_process: INT;
END_VAR

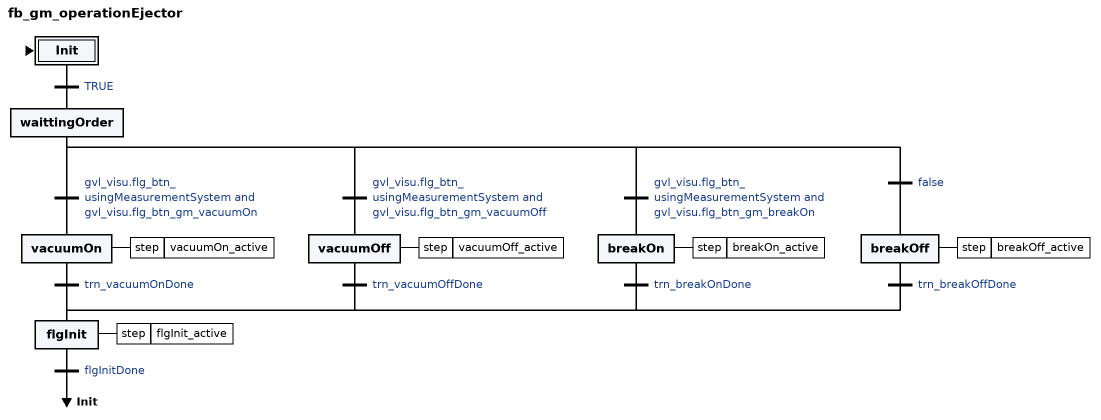
INITIAL_STEP Init:
END_STEP
TRANSITION FROM Init TO waittingOrder
    := TRUE;
END_TRANSITION
STEP waittingOrder:
END_STEP
TRANSITION FROM waittingOrder TO vacuumOn
    := gvl_visu.flg_btn_usingMeasurementSystem and gvl_visu.flg_btn_gm_vacuumOn;
END_TRANSITION
STEP vacuumOn:
    vacuumOn_active(N);  // step action
END_STEP
TRANSITION FROM vacuumOn TO flgInit
    := trn_vacuumOnDone;
END_TRANSITION
TRANSITION FROM waittingOrder TO vacuumOff
    := gvl_visu.flg_btn_usingMeasurementSystem and gvl_visu.flg_btn_gm_vacuumOff;
END_TRANSITION
STEP vacuumOff:
    vacuumOff_active(N);  // step action
END_STEP
TRANSITION FROM vacuumOff TO flgInit
    := trn_vacuumOffDone;
END_TRANSITION
TRANSITION FROM waittingOrder TO breakOn
    := gvl_visu.flg_btn_usingMeasurementSystem and gvl_visu.flg_btn_gm_breakOn;
END_TRANSITION
STEP breakOn:
    breakOn_active(N);  // step action
END_STEP
TRANSITION FROM breakOn TO flgInit
    := trn_breakOnDone;
END_TRANSITION
TRANSITION FROM waittingOrder TO breakOff
    := false;
END_TRANSITION
STEP breakOff:
    breakOff_active(N);  // step action
END_STEP
TRANSITION FROM breakOff TO flgInit
    := trn_breakOffDone;
END_TRANSITION
STEP flgInit:
    flgInit_active(N);  // step action
END_STEP
TRANSITION FROM flgInit TO Init
    := flgInitDone;
END_TRANSITION

ACTION breakOff_active:
IF breakOff._x AND breakOff.x = FALSE THEN
	trn_breakOffDone := FALSE;
	gvl_solv.fbi_gm_ejector.in_flg_run := FALSE;
	gvl_solv.fbi_gm_ejector.in_var_vacMode := eP_ejevacMode.breakOff;
	var_process := 0;
ELSIF breakOff._x AND breakOff.x THEN
	CASE var_process OF
		0:
			gvl_solv.fbi_gm_ejector.in_flg_run := TRUE;
			var_process := 0;
		1:
			IF gvl_solv.fbi_gm_ejector.out_flg_Done THEN
				gvl_solv.fbi_gm_ejector.in_flg_run := FALSE;
				trn_breakOffDone := TRUE;
			END_IF
	END_CASE
END_IF
END_ACTION

ACTION breakOn_active:
IF breakOn._x AND breakOn.x = FALSE THEN
	trn_breakOnDone := FALSE;
	gvl_solv.fbi_gm_ejector.in_flg_run := FALSE;
	gvl_solv.fbi_gm_ejector.in_var_vacMode := eP_ejevacMode.break;
	var_process := 0;
ELSIF breakOn._x AND breakOn._x THEN
	CASE var_process OF
		0:
			gvl_solv.fbi_gm_ejector.in_flg_run := TRUE;
			var_process := 1;
		1:
			IF gvl_solv.fbi_gm_ejector.out_flg_Done THEN
				gvl_solv.fbi_gm_ejector.in_flg_run := FALSE;
				trn_breakOnDone := TRUE;
			END_IF
	END_CASE
END_IF
END_ACTION

ACTION flgInit_active:
IF flgInit._x AND flgInit.x = FALSE THEN
	flgInitDone := FALSE;
	gvl_visu.flg_btn_gm_vacuumOn := FALSE;
	gvl_visu.flg_btn_gm_vacuumOff := FALSE;
	gvl_visu.flg_btn_gm_breakOn := FALSE;
	
ELSIF flgInit._x AND flgInit.x THEN
	flgInitDone := TRUE;
END_IF
END_ACTION

PROPERTY p_Init : bool
GET
p_init := THIS^.SFCInit;
END_GET
SET
THIS^.SFCInit := p_Init;
END_SET
END_PROPERTY

ACTION vacuumOff_active:
IF vacuumOff._x AND vacuumOff.x = FALSE THEN
	trn_vacuumOffDone := FALSE;
	gvl_solv.fbi_gm_ejector.in_flg_run := FALSE;
	gvl_solv.fbi_gm_ejector.in_var_vacMode := eP_ejevacMode.vacOff;
	var_process := 0;
ELSIF vacuumOff._x AND vacuumOff.x THEN
	CASE var_process OF
		0:
			gvl_solv.fbi_gm_ejector.in_flg_run := TRUE;
			var_process := 1;
		1:
			IF gvl_solv.fbi_gm_ejector.out_flg_Done THEN
			gvl_solv.fbi_gm_ejector.in_flg_run := FALSE;
			trn_vacuumOffDone := TRUE;
		END_IF
	END_CASE
END_IF
END_ACTION

ACTION vacuumOn_active:
IF vacuumOn._x AND vacuumOn.x = FALSE THEN
	trn_vacuumOnDone := FALSE;
	gvl_solv.fbi_gm_ejector.in_flg_run := FALSE;
	gvl_solv.fbi_gm_ejector.in_var_vacMode := eP_ejevacMode.halt;
	var_process := 0;
ELSIF vacuumOn._x AND vacuumOn.x THEN
	CASE var_process OF
		0:
			gvl_solv.fbi_gm_ejector.in_flg_run := TRUE;
			var_process := 1;
		1:
			IF gvl_solv.fbi_gm_ejector.out_flg_Done THEN
				gvl_solv.fbi_gm_ejector.in_flg_run := FALSE;
				trn_vacuumOnDone := TRUE;
			END_IF
	END_CASE
END_IF
END_ACTION

END_FUNCTION_BLOCK

// ---- FBs/fb_recordingSystem.TcPOU
FUNCTION_BLOCK fb_recordingSystem
VAR_INPUT
END_VAR
VAR_OUTPUT
END_VAR
VAR
	fbi_r_trigPalletize: R_TRIG;
	fbi_r_trigSample: R_TRIG;
	var_i: INT;
	fbi_r_trigP1: R_TRIG;
	fbi_r_trigP2: R_TRIG;
	fbi_r_trigP3: R_TRIG;
	var_buf_productNum: INT;
	var_scan: INT := 1;
	flg_productChanged: BOOL;
	var_scan2: INT;
	var_buf_cavNum: INT;
	var_scan3: INT := 1;
	var_buf_sapleCavNum: INT;
	flg_sampleCavChanged: BOOL;
	fbi_r_trigP4: R_TRIG;
END_VAR


	 CASE var_scan OF
		0:
		 	var_buf_productNum := gvl_param.var_currentProductID;
			var_scan := 1;
		1:
			IF var_buf_productNum <> gvl_param.var_currentProductID THEN
				flg_productChanged := TRUE;
				var_scan := 2;
			END_IF
		2:
			flg_productChanged := FALSE;
			var_scan := 0;
	 END_CASE
	 
	  CASE var_scan2 OF
		0:
		 	var_buf_cavNum := gvl_visu.var_in_cavNo;
			var_scan2 := 1;
		1:
			IF var_buf_cavNum <>  gvl_visu.var_in_cavNo THEN
				flg_productChanged := TRUE;
				var_scan2 := 2;
			END_IF
		2:
			flg_productChanged := FALSE;
			var_scan2 := 0;
	 END_CASE

	CASE var_scan3 OF
		0:
		 	var_buf_sapleCavNum := gvl_visu.var_in_sampleCavNo;
			var_scan3 := 1;
		1:
			IF var_buf_sapleCavNum <>  gvl_visu.var_in_sampleCavNo THEN
				flg_sampleCavChanged := TRUE;
				var_scan3 := 2;
			END_IF
		2:
			flg_sampleCavChanged := FALSE;
			var_scan3 := 0;
	 END_CASE

//saving triger
fbi_r_trigPalletize(CLK:=gvl_visu.flg_btn_savePalletize , Q=> );
fbi_r_trigSample(CLK:=gvl_visu.flg_btn_saveSample , Q=> );
//loading triger
fbi_r_trigP1(CLK:= gvl_param.var_currentTrayPos = 1 OR gvl_param.var_currentTrayPos = 2, 
				Q=> );
fbi_r_trigP3(CLK:=  flg_productChanged, 
				Q=> );
fbi_r_trigP4(CLK:=  flg_sampleCavChanged, 
				Q=> );
//save
IF fbi_r_trigPalletize.Q THEN
	FOR var_i := 1 TO 4 BY 1 DO
		gvl_param.var_productInfo[gvl_param.var_currentProductID].teachPos.palletize.upperLower[gvl_param.var_currentTrayPos].cav[gvl_visu.var_in_cavNo].Pos[var_i].x := gvl_visu.var_in_palletizePos.Pos[var_i].x;
		gvl_param.var_productInfo[gvl_param.var_currentProductID].teachPos.palletize.upperLower[gvl_param.var_currentTrayPos].cav[gvl_visu.var_in_cavNo].Pos[var_i].y := gvl_visu.var_in_palletizePos.Pos[var_i].y;
		gvl_param.var_productInfo[gvl_param.var_currentProductID].teachPos.palletize.upperLower[gvl_param.var_currentTrayPos].cav[gvl_visu.var_in_cavNo].Pos[var_i].z := gvl_visu.var_in_palletizePos.Pos[var_i].z;
	END_FOR
	gvl_param.var_productInfo[gvl_param.var_currentProductID].teachPos.initial.x := gvl_visu.var_in_initialPos.x;
	gvl_param.var_productInfo[gvl_param.var_currentProductID].teachPos.initial.y := gvl_visu.var_in_initialPos.y;
	gvl_param.var_productInfo[gvl_param.var_currentProductID].teachPos.initial.z := gvl_visu.var_in_initialPos.z;
	gvl_param.var_productInfo[gvl_param.var_currentProductID].teachPos.remove.x := gvl_visu.var_in_removePos.x;
	gvl_param.var_productInfo[gvl_param.var_currentProductID].teachPos.remove.y := gvl_visu.var_in_removePos.y;
	gvl_param.var_productInfo[gvl_param.var_currentProductID].teachPos.remove.z := gvl_visu.var_in_removePos.z;
	gvl_param.var_productInfo[gvl_param.var_currentProductID].teachPos.pickUp.x := gvl_visu.var_in_pickUpPos.x;
	gvl_param.var_productInfo[gvl_param.var_currentProductID].teachPos.pickUp.y := gvl_visu.var_in_pickUpPos.y;
	gvl_param.var_productInfo[gvl_param.var_currentProductID].teachPos.pickUp.z := gvl_visu.var_in_pickUpPos.z;
	gvl_param.var_productInfo[gvl_param.var_currentProductID].teachPos.palletize.upperLower[gvl_param.var_currentTrayPos].cav[gvl_visu.var_in_cavNo].teachingDetail.passingPos.x := gvl_visu.var_in_teachingDetail.passingPos.x;
	gvl_param.var_productInfo[gvl_param.var_currentProductID].teachPos.palletize.upperLower[gvl_param.var_currentTrayPos].cav[gvl_visu.var_in_cavNo].teachingDetail.passingPos.y := gvl_visu.var_in_teachingDetail.passingPos.y;
	gvl_param.var_productInfo[gvl_param.var_currentProductID].teachPos.palletize.upperLower[gvl_param.var_currentTrayPos].cav[gvl_visu.var_in_cavNo].teachingDetail.passingPos.z := gvl_visu.var_in_teachingDetail.passingPos.z;
	gvl_param.var_productInfo[gvl_param.var_currentProductID].teachPos.palletize.upperLower[gvl_param.var_currentTrayPos].cav[gvl_visu.var_in_cavNo].teachingDetail.settingPos.x := gvl_visu.var_in_teachingDetail.settingPos.x;
	gvl_param.var_productInfo[gvl_param.var_currentProductID].teachPos.palletize.upperLower[gvl_param.var_currentTrayPos].cav[gvl_visu.var_in_cavNo].teachingDetail.settingPos.y := gvl_visu.var_in_teachingDetail.settingPos.y;
	gvl_param.var_productInfo[gvl_param.var_currentProductID].teachPos.palletize.upperLower[gvl_param.var_currentTrayPos].cav[gvl_visu.var_in_cavNo].teachingDetail.settingPos.z := gvl_visu.var_in_teachingDetail.settingPos.z; 
	gvl_param.var_productInfo[gvl_param.var_currentProductID].teachPos.palletize.upperLower[gvl_param.var_currentTrayPos].cav[gvl_visu.var_in_cavNo].teachingDetailVels.x.vel := gvl_visu.var_in_teachingDetailVels.x.vel;
	gvl_param.var_productInfo[gvl_param.var_currentProductID].teachPos.palletize.upperLower[gvl_param.var_currentTrayPos].cav[gvl_visu.var_in_cavNo].teachingDetailVels.y.vel := gvl_visu.var_in_teachingDetailVels.y.vel;
	gvl_param.var_productInfo[gvl_param.var_currentProductID].teachPos.palletize.upperLower[gvl_param.var_currentTrayPos].cav[gvl_visu.var_in_cavNo].teachingDetailVels.z.vel := gvl_visu.var_in_teachingDetailVels.z.vel;
END_IF
IF fbi_r_trigSample.Q THEN
	gvl_param.var_productInfo[gvl_param.var_currentProductID].teachPos.sample[gvl_visu.var_in_sampleCavNo].x := gvl_visu.var_in_samplePos.x;
	gvl_param.var_productInfo[gvl_param.var_currentProductID].teachPos.sample[gvl_visu.var_in_sampleCavNo].y := gvl_visu.var_in_samplePos.y;
	gvl_param.var_productInfo[gvl_param.var_currentProductID].teachPos.sample[gvl_visu.var_in_sampleCavNo].z := gvl_visu.var_in_samplePos.z;
END_IF

//load
IF fbi_r_trigP1.Q OR fbi_r_trigP3.Q THEN
	FOR var_i := 1 TO 4 BY 1 DO
		gvl_visu.var_in_palletizePos.Pos[var_i].x :=gvl_param.var_productInfo[gvl_param.var_currentProductID].teachPos.palletize.upperLower[gvl_param.var_currentTrayPos].cav[gvl_visu.var_in_cavNo].Pos[var_i].x;
		gvl_visu.var_in_palletizePos.Pos[var_i].y :=gvl_param.var_productInfo[gvl_param.var_currentProductID].teachPos.palletize.upperLower[gvl_param.var_currentTrayPos].cav[gvl_visu.var_in_cavNo].Pos[var_i].y;
		gvl_visu.var_in_palletizePos.Pos[var_i].z :=gvl_param.var_productInfo[gvl_param.var_currentProductID].teachPos.palletize.upperLower[gvl_param.var_currentTrayPos].cav[gvl_visu.var_in_cavNo].Pos[var_i].z;
	END_FOR
	gvl_visu.var_in_initialPos.x := gvl_param.var_productInfo[gvl_param.var_currentProductID].teachPos.initial.x;
	gvl_visu.var_in_initialPos.y := gvl_param.var_productInfo[gvl_param.var_currentProductID].teachPos.initial.y;
	gvl_visu.var_in_initialPos.z := gvl_param.var_productInfo[gvl_param.var_currentProductID].teachPos.initial.z;
	gvl_visu.var_in_removePos.x := gvl_param.var_productInfo[gvl_param.var_currentProductID].teachPos.remove.x;
	gvl_visu.var_in_removePos.y := gvl_param.var_productInfo[gvl_param.var_currentProductID].teachPos.remove.y;
	gvl_visu.var_in_removePos.z := gvl_param.var_productInfo[gvl_param.var_currentProductID].teachPos.remove.z;
	gvl_visu.var_in_pickUpPos.x := gvl_param.var_productInfo[gvl_param.var_currentProductID].teachPos.pickUp.x;
	gvl_visu.var_in_pickUpPos.y := gvl_param.var_productInfo[gvl_param.var_currentProductID].teachPos.pickUp.y;
	gvl_visu.var_in_pickUpPos.z := gvl_param.var_productInfo[gvl_param.var_currentProductID].teachPos.pickUp.z;
	gvl_visu.var_in_teachingDetail.passingPos.x := gvl_param.var_productInfo[gvl_param.var_currentProductID].teachPos.palletize.upperLower[gvl_param.var_currentTrayPos].cav[gvl_visu.var_in_cavNo].teachingDetail.passingPos.x;
	gvl_visu.var_in_teachingDetail.passingPos.y := gvl_param.var_productInfo[gvl_param.var_currentProductID].teachPos.palletize.upperLower[gvl_param.var_currentTrayPos].cav[gvl_visu.var_in_cavNo].teachingDetail.passingPos.y;
	gvl_visu.var_in_teachingDetail.passingPos.z := gvl_param.var_productInfo[gvl_param.var_currentProductID].teachPos.palletize.upperLower[gvl_param.var_currentTrayPos].cav[gvl_visu.var_in_cavNo].teachingDetail.passingPos.z;
	gvl_visu.var_in_teachingDetail.settingPos.x := gvl_param.var_productInfo[gvl_param.var_currentProductID].teachPos.palletize.upperLower[gvl_param.var_currentTrayPos].cav[gvl_visu.var_in_cavNo].teachingDetail.settingPos.x;
	gvl_visu.var_in_teachingDetail.settingPos.y := gvl_param.var_productInfo[gvl_param.var_currentProductID].teachPos.palletize.upperLower[gvl_param.var_currentTrayPos].cav[gvl_visu.var_in_cavNo].teachingDetail.settingPos.y;
	gvl_visu.var_in_teachingDetail.settingPos.z := gvl_param.var_productInfo[gvl_param.var_currentProductID].teachPos.palletize.upperLower[gvl_param.var_currentTrayPos].cav[gvl_visu.var_in_cavNo].teachingDetail.settingPos.z;
	gvl_visu.var_in_teachingDetailVels.x.vel := gvl_param.var_productInfo[gvl_param.var_currentProductID].teachPos.palletize.upperLower[gvl_param.var_currentTrayPos].cav[gvl_visu.var_in_cavNo].teachingDetailVels.x.vel;
	gvl_visu.var_in_teachingDetailVels.y.vel := gvl_param.var_productInfo[gvl_param.var_currentProductID].teachPos.palletize.upperLower[gvl_param.var_currentTrayPos].cav[gvl_visu.var_in_cavNo].teachingDetailVels.y.vel;
	gvl_visu.var_in_teachingDetailVels.z.vel := gvl_param.var_productInfo[gvl_param.var_currentProductID].teachPos.palletize.upperLower[gvl_param.var_currentTrayPos].cav[gvl_visu.var_in_cavNo].teachingDetailVels.z.vel;
END_IF
IF  fbi_r_trigP3.Q OR fbi_r_trigP4.Q THEN
	gvl_visu.var_in_samplePos.x := gvl_param.var_productInfo[gvl_param.var_currentProductID].teachPos.sample[gvl_visu.var_in_sampleCavNo].x;
	gvl_visu.var_in_samplePos.y := gvl_param.var_productInfo[gvl_param.var_currentProductID].teachPos.sample[gvl_visu.var_in_sampleCavNo].y;
	gvl_visu.var_in_samplePos.z := gvl_param.var_productInfo[gvl_param.var_currentProductID].teachPos.sample[gvl_visu.var_in_sampleCavNo].z;
END_IF

END_FUNCTION_BLOCK

// ---- FBs/fb_productGenerator.TcPOU
FUNCTION_BLOCK fb_productGenerator
VAR_INPUT
END_VAR
VAR_OUTPUT
END_VAR
VAR 
	fbi_r_trigSave: R_TRIG;
	var_scan: INT;
	var_buf_productNnum: INT;
END_VAR

fbi_r_trigSave(CLK:=gvl_visu.flg_btn_saveProductInfo , Q=> );
//load
CASE var_scan OF
	0:
		var_buf_productNnum := gvl_param.var_productInfo[gvl_visu.var_in_productGenerate.num].num;
		var_scan := 1;
	1:
		IF var_buf_productNnum <> gvl_param.var_productInfo[gvl_visu.var_in_productGenerate.num].num THEN
			gvl_visu.var_in_productGenerate.num					:= gvl_param.var_productInfo[gvl_visu.var_in_productGenerate.num].num;
			gvl_visu.var_in_productGenerate.name				:= gvl_param.var_productInfo[gvl_visu.var_in_productGenerate.num].name;
			gvl_visu.var_in_productGenerate.bottomPocketQty		:= gvl_param.var_productInfo[gvl_visu.var_in_productGenerate.num].bottomPocketQty;
			gvl_visu.var_in_productGenerate.vertivalPocketQty	:= gvl_param.var_productInfo[gvl_visu.var_in_productGenerate.num].vertivalPocketQty;
			gvl_visu.var_in_productGenerate.pocketSumQty		:= gvl_param.var_productInfo[gvl_visu.var_in_productGenerate.num].pocketSumQty;
			gvl_visu.var_in_productGenerate.startCav			:= gvl_param.var_productInfo[gvl_visu.var_in_productGenerate.num].startCav;
			gvl_visu.var_in_productGenerate.cavQty				:= gvl_param.var_productInfo[gvl_visu.var_in_productGenerate.num].cavQty;
			gvl_visu.var_in_productGenerate.gateLength_max		:= gvl_param.var_productInfo[gvl_visu.var_in_productGenerate.num].gateLength_max;
			gvl_visu.var_in_productGenerate.gateLength_min		:= gvl_param.var_productInfo[gvl_visu.var_in_productGenerate.num].gateLength_min;
			gvl_visu.var_in_productGenerate.autoVels.x.vel		:= gvl_param.var_productInfo[gvl_visu.var_in_productGenerate.num].autoVels.x.vel;
			gvl_visu.var_in_productGenerate.autoVels.x.acc		:= gvl_param.var_productInfo[gvl_visu.var_in_productGenerate.num].autoVels.x.acc;
			gvl_visu.var_in_productGenerate.autoVels.x.dcc		:= gvl_param.var_productInfo[gvl_visu.var_in_productGenerate.num].autoVels.x.dcc;
			gvl_visu.var_in_productGenerate.autoVels.y.vel		:= gvl_param.var_productInfo[gvl_visu.var_in_productGenerate.num].autoVels.y.vel;
			gvl_visu.var_in_productGenerate.autoVels.y.acc		:= gvl_param.var_productInfo[gvl_visu.var_in_productGenerate.num].autoVels.y.acc;
			gvl_visu.var_in_productGenerate.autoVels.y.dcc		:= gvl_param.var_productInfo[gvl_visu.var_in_productGenerate.num].autoVels.y.dcc;
			gvl_visu.var_in_productGenerate.autoVels.z.vel		:= gvl_param.var_productInfo[gvl_visu.var_in_productGenerate.num].autoVels.z.vel;
			gvl_visu.var_in_productGenerate.autoVels.z.acc		:= gvl_param.var_productInfo[gvl_visu.var_in_productGenerate.num].autoVels.z.acc;
			gvl_visu.var_in_productGenerate.autoVels.z.dcc		:= gvl_param.var_productInfo[gvl_visu.var_in_productGenerate.num].autoVels.z.dcc;
			gvl_visu.var_in_productGenerate.manaulVels.x.vel	:= gvl_param.var_productInfo[gvl_visu.var_in_productGenerate.num].manaulVels.x.vel;
			gvl_visu.var_in_productGenerate.manaulVels.y.vel	:= gvl_param.var_productInfo[gvl_visu.var_in_productGenerate.num].manaulVels.y.vel;
			gvl_visu.var_in_productGenerate.manaulVels.z.vel	:= gvl_param.var_productInfo[gvl_visu.var_in_productGenerate.num].manaulVels.z.vel;
			gvl_visu.var_in_productGenerate.incjetMsgNo			:= gvl_param.var_productInfo[gvl_visu.var_in_productGenerate.num].incjetMsgNo;
			gvl_visu.var_in_productGenerate.flg_mode_measurement:= gvl_param.var_productInfo[gvl_visu.var_in_productGenerate.num].flg_mode_measurement;
			gvl_visu.var_in_productGenerate.flg_mode_stocker	:= gvl_param.var_productInfo[gvl_visu.var_in_productGenerate.num].flg_mode_stocker;
			var_scan := 2;
		END_IF
	2:
		var_scan := 0;
END_CASE
//save
IF fbi_r_trigSave.Q THEN
	gvl_param.var_productInfo[gvl_visu.var_in_productGenerate.num].num					:= gvl_visu.var_in_productGenerate.num;
	gvl_param.var_productInfo[gvl_visu.var_in_productGenerate.num].name					:= gvl_visu.var_in_productGenerate.name;
	gvl_visu.var_in_currentProduct[gvl_visu.var_in_productGenerate.num]					:= gvl_visu.var_in_productGenerate.name;
	gvl_param.var_productInfo[gvl_visu.var_in_productGenerate.num].bottomPocketQty		:= gvl_visu.var_in_productGenerate.bottomPocketQty;
	gvl_param.var_productInfo[gvl_visu.var_in_productGenerate.num].vertivalPocketQty	:= gvl_visu.var_in_productGenerate.vertivalPocketQty;
	gvl_param.var_productInfo[gvl_visu.var_in_productGenerate.num].pocketSumQty			:= gvl_visu.var_in_productGenerate.bottomPocketQty * gvl_visu.var_in_productGenerate.vertivalPocketQty;
	gvl_param.var_productInfo[gvl_visu.var_in_productGenerate.num].startCav				:= gvl_visu.var_in_productGenerate.startCav;
	gvl_param.var_productInfo[gvl_visu.var_in_productGenerate.num].cavQty				:= gvl_visu.var_in_productGenerate.cavQty;
	gvl_param.var_productInfo[gvl_visu.var_in_productGenerate.num].gateLength_max		:= gvl_visu.var_in_productGenerate.gateLength_max;
	gvl_param.var_productInfo[gvl_visu.var_in_productGenerate.num].gateLength_min		:= gvl_visu.var_in_productGenerate.gateLength_min;
	gvl_param.var_productInfo[gvl_visu.var_in_productGenerate.num].autoVels.x.vel		:= gvl_visu.var_in_productGenerate.autoVels.x.vel;
	gvl_param.var_productInfo[gvl_visu.var_in_productGenerate.num].autoVels.x.acc		:= gvl_visu.var_in_productGenerate.autoVels.x.acc;
	gvl_param.var_productInfo[gvl_visu.var_in_productGenerate.num].autoVels.x.dcc		:= gvl_visu.var_in_productGenerate.autoVels.x.dcc;
	gvl_param.var_productInfo[gvl_visu.var_in_productGenerate.num].autoVels.y.vel		:= gvl_visu.var_in_productGenerate.autoVels.y.vel;
	gvl_param.var_productInfo[gvl_visu.var_in_productGenerate.num].autoVels.y.acc		:= gvl_visu.var_in_productGenerate.autoVels.y.acc;
	gvl_param.var_productInfo[gvl_visu.var_in_productGenerate.num].autoVels.y.dcc		:= gvl_visu.var_in_productGenerate.autoVels.y.dcc;
	gvl_param.var_productInfo[gvl_visu.var_in_productGenerate.num].autoVels.z.vel		:= gvl_visu.var_in_productGenerate.autoVels.z.vel;
	gvl_param.var_productInfo[gvl_visu.var_in_productGenerate.num].autoVels.z.acc		:= gvl_visu.var_in_productGenerate.autoVels.z.acc;
	gvl_param.var_productInfo[gvl_visu.var_in_productGenerate.num].autoVels.z.dcc		:= gvl_visu.var_in_productGenerate.autoVels.z.dcc;
	gvl_param.var_productInfo[gvl_visu.var_in_productGenerate.num].manaulVels.x.vel		:= gvl_visu.var_in_productGenerate.manaulVels.x.vel;
	gvl_param.var_productInfo[gvl_visu.var_in_productGenerate.num].manaulVels.y.vel		:= gvl_visu.var_in_productGenerate.manaulVels.y.vel;
	gvl_param.var_productInfo[gvl_visu.var_in_productGenerate.num].manaulVels.z.vel		:= gvl_visu.var_in_productGenerate.manaulVels.z.vel;
	gvl_param.var_productInfo[gvl_visu.var_in_productGenerate.num].incjetMsgNo			:= gvl_visu.var_in_productGenerate.incjetMsgNo;
	gvl_param.var_productInfo[gvl_visu.var_in_productGenerate.num].flg_mode_measurement	:= gvl_visu.var_in_productGenerate.flg_mode_measurement;
	gvl_param.var_productInfo[gvl_visu.var_in_productGenerate.num].flg_mode_stocker		:= gvl_visu.var_in_productGenerate.flg_mode_stocker;
END_IF

END_FUNCTION_BLOCK

// ---- FBs/gateMeasurementModule/fb_gm_operationSV.TcPOU
FUNCTION_BLOCK fb_gm_operationSV
VAR_INPUT
END_VAR
VAR_OUTPUT
END_VAR
VAR
	trn_gm_chuckOpenDone: BOOL;
	trn_gm_chuckCloseDone: BOOL;
	trn_gm_pushCloseDone: BOOL;
	trn_gm_pushOpenDone: BOOL;
	trn_gm_rotaryOriginDone: BOOL;
	trn_gm_rotaryMovingDone: BOOL;
	trn_gm_pickUpOriginDone: BOOL;
	trn_gm_pickUpMovingDone: BOOL;
	trn_gm_stampOriginDone: BOOL;
	trn_gm_stampMovingDone: BOOL;
	trn_flgInitDone: BOOL;
	flg_test: BOOL;
	flg_test2: BOOL;
END_VAR

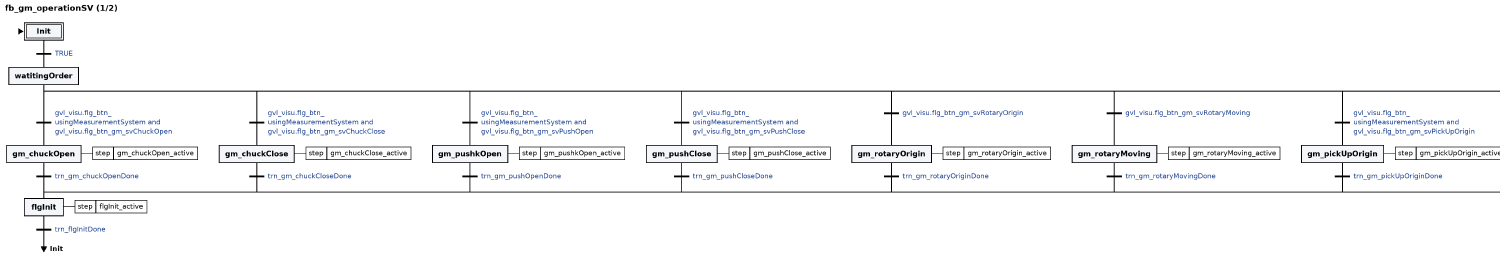
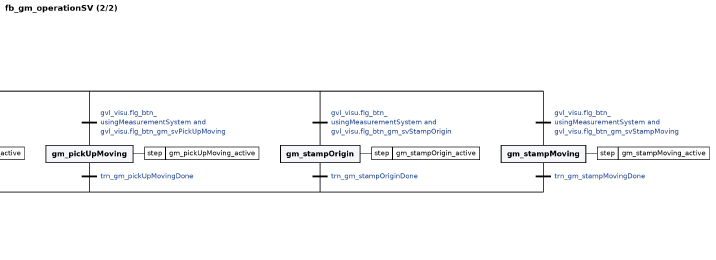
INITIAL_STEP Init:
END_STEP
TRANSITION FROM Init TO watitingOrder
    := TRUE;
END_TRANSITION
STEP watitingOrder:
END_STEP
TRANSITION FROM watitingOrder TO gm_chuckOpen
    := gvl_visu.flg_btn_usingMeasurementSystem and gvl_visu.flg_btn_gm_svChuckOpen;
END_TRANSITION
STEP gm_chuckOpen:
    gm_chuckOpen_active(N);  // step action
END_STEP
TRANSITION FROM gm_chuckOpen TO flgInit
    := trn_gm_chuckOpenDone;
END_TRANSITION
TRANSITION FROM watitingOrder TO gm_chuckClose
    := gvl_visu.flg_btn_usingMeasurementSystem and gvl_visu.flg_btn_gm_svChuckClose;
END_TRANSITION
STEP gm_chuckClose:
    gm_chuckClose_active(N);  // step action
END_STEP
TRANSITION FROM gm_chuckClose TO flgInit
    := trn_gm_chuckCloseDone;
END_TRANSITION
TRANSITION FROM watitingOrder TO gm_pushkOpen
    := gvl_visu.flg_btn_usingMeasurementSystem and gvl_visu.flg_btn_gm_svPushOpen;
END_TRANSITION
STEP gm_pushkOpen:
    gm_pushkOpen_active(N);  // step action
END_STEP
TRANSITION FROM gm_pushkOpen TO flgInit
    := trn_gm_pushOpenDone;
END_TRANSITION
TRANSITION FROM watitingOrder TO gm_pushClose
    := gvl_visu.flg_btn_usingMeasurementSystem and gvl_visu.flg_btn_gm_svPushClose;
END_TRANSITION
STEP gm_pushClose:
    gm_pushClose_active(N);  // step action
END_STEP
TRANSITION FROM gm_pushClose TO flgInit
    := trn_gm_pushCloseDone;
END_TRANSITION
TRANSITION FROM watitingOrder TO gm_rotaryOrigin
    := gvl_visu.flg_btn_gm_svRotaryOrigin;
END_TRANSITION
STEP gm_rotaryOrigin:
    gm_rotaryOrigin_active(N);  // step action
END_STEP
TRANSITION FROM gm_rotaryOrigin TO flgInit
    := trn_gm_rotaryOriginDone;
END_TRANSITION
TRANSITION FROM watitingOrder TO gm_rotaryMoving
    := gvl_visu.flg_btn_gm_svRotaryMoving;
END_TRANSITION
STEP gm_rotaryMoving:
    gm_rotaryMoving_active(N);  // step action
END_STEP
TRANSITION FROM gm_rotaryMoving TO flgInit
    := trn_gm_rotaryMovingDone;
END_TRANSITION
TRANSITION FROM watitingOrder TO gm_pickUpOrigin
    := gvl_visu.flg_btn_usingMeasurementSystem and gvl_visu.flg_btn_gm_svPickUpOrigin;
END_TRANSITION
STEP gm_pickUpOrigin:
    gm_pickUpOrigin_active(N);  // step action
END_STEP
TRANSITION FROM gm_pickUpOrigin TO flgInit
    := trn_gm_pickUpOriginDone;
END_TRANSITION
TRANSITION FROM watitingOrder TO gm_pickUpMoving
    := gvl_visu.flg_btn_usingMeasurementSystem and gvl_visu.flg_btn_gm_svPickUpMoving;
END_TRANSITION
STEP gm_pickUpMoving:
    gm_pickUpMoving_active(N);  // step action
END_STEP
TRANSITION FROM gm_pickUpMoving TO flgInit
    := trn_gm_pickUpMovingDone;
END_TRANSITION
TRANSITION FROM watitingOrder TO gm_stampOrigin
    := gvl_visu.flg_btn_usingMeasurementSystem and gvl_visu.flg_btn_gm_svStampOrigin;
END_TRANSITION
STEP gm_stampOrigin:
    gm_stampOrigin_active(N);  // step action
END_STEP
TRANSITION FROM gm_stampOrigin TO flgInit
    := trn_gm_stampOriginDone;
END_TRANSITION
TRANSITION FROM watitingOrder TO gm_stampMoving
    := gvl_visu.flg_btn_usingMeasurementSystem and gvl_visu.flg_btn_gm_svStampMoving;
END_TRANSITION
STEP gm_stampMoving:
    gm_stampMoving_active(N);  // step action
END_STEP
TRANSITION FROM gm_stampMoving TO flgInit
    := trn_gm_stampMovingDone;
END_TRANSITION
STEP flgInit:
    flgInit_active(N);  // step action
END_STEP
TRANSITION FROM flgInit TO Init
    := trn_flgInitDone;
END_TRANSITION

ACTION flgInit_active:
IF flgInit._x AND flgInit.x = FALSE THEN
	trn_flgInitDone := FALSE;
	gvl_visu.flg_btn_gm_svChuckOpen := FALSE;
	gvl_visu.flg_btn_gm_svChuckClose := FALSE;
	gvl_visu.flg_btn_gm_svPushOpen := FALSE;
	gvl_visu.flg_btn_gm_svPushClose := FALSE;
	gvl_visu.flg_btn_gm_svRotaryOrigin := FALSE;
	gvl_visu.flg_btn_gm_svRotaryMoving := FALSE;
	gvl_visu.flg_btn_gm_svPickUpOrigin := FALSE;
	gvl_visu.flg_btn_gm_svPickUpMoving := FALSE;
	gvl_visu.flg_btn_gm_svStampOrigin := FALSE;
	gvl_visu.flg_btn_gm_svStampMoving := FALSE;
ELSIF flgInit._x AND flgInit.x THEN
	trn_flgInitDone := TRUE;
END_IF
END_ACTION

ACTION gm_chuckClose_active:
IF gm_chuckClose._x AND gm_chuckClose.x = FALSE THEN
	trn_gm_chuckCloseDone := FALSE;
	gvl_solv.fbi_gm_chuck.in_flg_run := FALSE;
	gvl_solv.fbi_gm_chuck.in_var_moveMode := eP_svMoveMode.svB;
ELSIF gm_chuckClose._x AND gm_chuckClose.x THEN
	gvl_solv.fbi_gm_chuck.in_flg_run := TRUE;
	IF gvl_solv.fbi_gm_chuck.out_flg_Done THEN
		gvl_solv.fbi_gm_chuck.in_flg_run := FALSE;
		trn_gm_chuckCloseDone := TRUE;
	END_IF
END_IF
END_ACTION

ACTION gm_chuckOpen_active:
IF gm_chuckOpen._x AND gm_chuckOpen.x = FALSE THEN
	trn_gm_chuckOpenDone := FALSE;
	gvl_solv.fbi_gm_chuck.in_flg_run := FALSE;
	gvl_solv.fbi_gm_chuck.in_var_moveMode := eP_svMoveMode.svA;
ELSIF gm_chuckOpen._x AND gm_chuckOpen.x THEN
	gvl_solv.fbi_gm_chuck.in_flg_run := TRUE;
	IF gvl_solv.fbi_gm_chuck.out_flg_Done THEN
		gvl_solv.fbi_gm_chuck.in_flg_run := FALSE;
		trn_gm_chuckOpenDone := TRUE;
	END_IF
END_IF
END_ACTION

ACTION gm_pickUpMoving_active:
IF gm_pickUpMoving._x AND gm_pickUpMoving.x = FALSE THEN
	trn_gm_pickUpMovingDone := FALSE;
	gvl_solv.fbi_gm_pickup.in_flg_run := FALSE;
	gvl_solv.fbi_gm_pickup.in_var_moveMode := eP_svMoveMode.svB;
ELSIF gm_pickUpMoving._x AND gm_pickUpMoving.x THEN
		gvl_solv.fbi_gm_pickup.in_flg_run := TRUE;
	IF gvl_solv.fbi_gm_pickup.out_flg_Done THEN
		gvl_solv.fbi_gm_pickup.in_flg_run := FALSE;
		trn_gm_pickUpMovingDone := TRUE;
	END_IF
END_IF
END_ACTION

ACTION gm_pickUpOrigin_active:
IF gm_pickUpOrigin._x AND gm_pickUpOrigin.x = FALSE THEN
	trn_gm_pickUpOriginDone := FALSE;
	gvl_solv.fbi_gm_pickup.in_flg_run := FALSE;
	gvl_solv.fbi_gm_pickup.in_var_moveMode := eP_svMoveMode.svA;
ELSIF gm_pickUpOrigin._x AND gm_pickUpOrigin.x THEN
		gvl_solv.fbi_gm_pickup.in_flg_run := TRUE;
	IF gvl_solv.fbi_gm_pickup.out_flg_Done THEN
		gvl_solv.fbi_gm_pickup.in_flg_run := FALSE;
		trn_gm_pickUpOriginDone := TRUE;
	END_IF
END_IF
END_ACTION

ACTION gm_pushClose_active:
IF gm_pushClose._x AND gm_pushClose.x = FALSE THEN
	trn_gm_pushCloseDone := FALSE;
	gvl_solv.fbi_gm_push.in_flg_run := FALSE;
	gvl_solv.fbi_gm_push.in_var_moveMode := eP_svMoveMode.svB;
ELSIF gm_pushClose._x AND gm_pushClose.x THEN
	gvl_solv.fbi_gm_push.in_flg_run := TRUE;
	IF gvl_solv.fbi_gm_push.out_flg_Done THEN
		gvl_solv.fbi_gm_push.in_flg_run := FALSE;
		trn_gm_pushCloseDone := TRUE;
	END_IF
END_IF
END_ACTION

ACTION gm_pushkOpen_active:
IF gm_pushkOpen._x AND gm_pushkOpen.x = FALSE THEN
	trn_gm_pushOpenDone := FALSE;
	gvl_solv.fbi_gm_push.in_flg_run := FALSE;
	gvl_solv.fbi_gm_push.in_var_moveMode := eP_svMoveMode.svA;
ELSIF gm_pushkOpen._x AND gm_pushkOpen.x THEN
	gvl_solv.fbi_gm_push.in_flg_run := TRUE;
	IF gvl_solv.fbi_gm_push.out_flg_Done THEN
 		gvl_solv.fbi_gm_push.in_flg_run := FALSE;
		trn_gm_pushOpenDone := TRUE;
	END_IF
END_IF
END_ACTION

ACTION gm_rotaryMoving_active:
IF gm_rotaryMoving._x AND gm_rotaryMoving.x = FALSE THEN
	trn_gm_rotaryMovingDone := FALSE;
	gvl_solv.fbi_gm_rotary.in_flg_run := FALSE;
	gvl_solv.fbi_gm_rotary.in_var_moveMode := eP_svMoveMode.svB;
ELSIF gm_rotaryMoving._x AND gm_rotaryMoving.x THEN
		gvl_solv.fbi_gm_rotary.in_flg_run := TRUE;
	IF gvl_solv.fbi_gm_rotary.out_flg_Done THEN
		gvl_solv.fbi_gm_rotary.in_flg_run := FALSE;
		trn_gm_rotaryMovingDone := TRUE;
	END_IF
END_IF
END_ACTION

ACTION gm_rotaryOrigin_active:
IF gm_rotaryOrigin._x AND gm_rotaryOrigin.x = FALSE THEN
	trn_gm_rotaryOriginDone := FALSE;
	gvl_solv.fbi_gm_rotary.in_flg_run := FALSE;
	gvl_solv.fbi_gm_rotary.in_var_moveMode := eP_svMoveMode.svA;
ELSIF gm_rotaryOrigin._x AND gm_rotaryOrigin.x THEN
	gvl_solv.fbi_gm_rotary.in_flg_run := TRUE;
	IF gvl_solv.fbi_gm_rotary.out_flg_Done THEN
		gvl_solv.fbi_gm_rotary.in_flg_run := FALSE;
		trn_gm_rotaryOriginDone := TRUE;
	END_IF
END_IF
END_ACTION

ACTION gm_stampMoving_active:
IF gm_stampMoving._x AND gm_stampMoving.x = FALSE THEN
	trn_gm_stampMovingDone := FALSE;
	gvl_solv.fbi_gm_stamp.in_flg_run := FALSE;
	gvl_solv.fbi_gm_stamp.in_var_moveMode := eP_svMoveMode.svB;
ELSIF gm_stampMoving._x AND gm_stampMoving.x THEN
		gvl_solv.fbi_gm_stamp.in_flg_run := TRUE;
	IF gvl_solv.fbi_gm_stamp.out_flg_Done THEN
		gvl_solv.fbi_gm_stamp.in_flg_run := FALSE;
		trn_gm_stampMovingDone := TRUE;
	END_IF
END_IF
END_ACTION

ACTION gm_stampOrigin_active:
IF gm_stampOrigin._x AND gm_stampOrigin.x = FALSE THEN
	trn_gm_stampOriginDone := FALSE;
	gvl_solv.fbi_gm_stamp.in_flg_run := FALSE;
	gvl_solv.fbi_gm_stamp.in_var_moveMode := eP_svMoveMode.svA;
ELSIF gm_stampOrigin._x AND gm_stampOrigin.x THEN
		gvl_solv.fbi_gm_stamp.in_flg_run := TRUE;
	IF gvl_solv.fbi_gm_stamp.out_flg_Done THEN
		gvl_solv.fbi_gm_stamp.in_flg_run := FALSE;
		trn_gm_stampOriginDone := TRUE;
	END_IF
END_IF
END_ACTION

PROPERTY p_Init : bool
GET
p_init := THIS^.SFCInit;
END_GET
SET
THIS^.SFCInit := p_init;
END_SET
END_PROPERTY

END_FUNCTION_BLOCK

// ---- FBs/gateMeasurementModule/fb_gm_setting.TcPOU
FUNCTION_BLOCK fb_gm_setting
VAR_INPUT
END_VAR
VAR_OUTPUT
END_VAR
VAR
	var_scan: INT := 1;
	var_buf_productID: INT;
	flg_productChanged: BOOL;
END_VAR

//vels
gvl_gm.var_buf_manualVel := gvl_visu.var_gm_manualRotaryVel;
gvl_gm.var_buf_autoVel := gvl_visu.var_gm_autoRotaryVel;
gvl_gm.var_buf_autoAcc := gvl_visu.var_gm_autoRotaryAcc;
gvl_gm.var_buf_autoDec := gvl_visu.var_gm_autoRotaryDec;
//jog
gvl_axis.fbi_mc_jogR.Position := gvl_visu.var_gm_rotaryInch;
CASE gvl_visu.var_radio_rotaryJogMode OF
	0:
		gvl_axis.fbi_mc_jogR.Mode := E_JogMode.MC_JOGMODE_INCHING;
	1:
		gvl_axis.fbi_mc_jogR.Mode := E_JogMode.MC_JOGMODE_CONTINOUS;
END_CASE

IF gvl_visu.flg_btn_rotaryRigt THEN
	gvl_axis.fbi_mc_jogR.JogForward := TRUE;
ELSIF gvl_visu.flg_btn_rotaryLeft THEN
	gvl_axis.fbi_mc_jogR.JogBackwards := TRUE;
ELSE
	gvl_axis.fbi_mc_jogR.JogForward := FALSE;
	gvl_axis.fbi_mc_jogR.JogBackwards := FALSE;
END_IF

//recording position

IF gvl_visu.flg_btn_rotaryPos THEN
	gvl_param.var_productInfo[gvl_param.var_currentProductID].teachPos.gm_rotary.origin := gvl_visu.var_rotaryPos.origin;
	gvl_param.var_productInfo[gvl_param.var_currentProductID].teachPos.gm_rotary.pickUp := gvl_visu.var_rotaryPos.pickUp;
	gvl_param.var_productInfo[gvl_param.var_currentProductID].teachPos.gm_rotary.set := gvl_visu.var_rotaryPos.set;
	gvl_param.var_productInfo[gvl_param.var_currentProductID].teachPos.gm_rotary.remove := gvl_visu.var_rotaryPos.remove;
END_IF


IF flg_productChanged THEN
	gvl_visu.var_rotaryPos.origin := gvl_param.var_productInfo[gvl_param.var_currentProductID].teachPos.gm_rotary.origin;
	gvl_visu.var_rotaryPos.pickUp := gvl_param.var_productInfo[gvl_param.var_currentProductID].teachPos.gm_rotary.pickUp;
	gvl_visu.var_rotaryPos.set := gvl_param.var_productInfo[gvl_param.var_currentProductID].teachPos.gm_rotary.set;
	gvl_visu.var_rotaryPos.remove := gvl_param.var_productInfo[gvl_param.var_currentProductID].teachPos.gm_rotary.remove;
END_IF



CASE var_scan OF
		0:
		 	var_buf_productID := gvl_param.var_currentProductID;
			var_scan := 1;
		1:
			IF var_buf_productID <> gvl_param.var_currentProductID THEN
				flg_productChanged := TRUE;
				var_scan := 2;
			END_IF
		2:
			flg_productChanged := FALSE;
			var_scan := 0;
END_CASE

END_FUNCTION_BLOCK

// ---- FBs/gateMeasurementModule/fb_gm_PTP.TcPOU
FUNCTION_BLOCK fb_gm_PTP
VAR_INPUT
	in_flg_run : bool;
END_VAR
VAR_OUTPUT
END_VAR
VAR
	var_process: INT;
END_VAR

IF NOT in_flg_run THEN
	var_process := 0;
END_IF
CASE var_process OF
	0:
		gvl_axis.ref_r.Execute := FALSE;
		var_process := 1;
	1:
		IF gvl_visu.flg_btn_gm_moveOrigin THEN
			gvl_axis.ref_r.Position := gvl_param.var_productInfo[gvl_param.var_currentProductID].teachPos.gm_rotary.origin;
			var_process := 2;
		ELSIF gvl_visu.flg_btn_gm_movePickUp THEN
			gvl_axis.ref_r.Position := gvl_param.var_productInfo[gvl_param.var_currentProductID].teachPos.gm_rotary.pickUp;
			var_process := 2;
		ELSIF gvl_visu.flg_btn_gm_moveSet THEN
			gvl_axis.ref_r.Position := gvl_param.var_productInfo[gvl_param.var_currentProductID].teachPos.gm_rotary.set;
			var_process := 2;
		ELSIF gvl_visu.flg_btn_gm_moveRemove THEN
			gvl_axis.ref_r.Position := gvl_param.var_productInfo[gvl_param.var_currentProductID].teachPos.gm_rotary.remove;
			var_process := 2;
		END_IF
	2:
		gvl_axis.ref_r.Execute := TRUE;
		IF gvl_axis.ref_r.Error THEN
			var_process := 0;
		END_IF
		IF gvl_axis.ref_r.Done THEN
			gvl_axis.ref_r.Execute := FALSE;
			var_process := 0;
		END_IF
END_CASE

END_FUNCTION_BLOCK

// ---- FBs/fb_debugData.TcPOU
FUNCTION_BLOCK fb_debugData
VAR_INPUT
END_VAR
VAR_OUTPUT
END_VAR
VAR
	productID: INT;
END_VAR

productID := 0;


gvl_param.var_productInfo[productID].name 				:= '---ForDebug---';
gvl_param.var_productInfo[productID].num				:= productID;
gvl_param.var_productInfo[productID].bottomPocketQty 	:= 5;
gvl_param.var_productInfo[productID].vertivalPocketQty 	:= 3;
gvl_param.var_productInfo[productID].startCav 			:= 1;
gvl_param.var_productInfo[productID].cavQty 			:= 8;
gvl_param.var_productInfo[productID].gateLength_max 	:= 30000;
gvl_param.var_productInfo[productID].gateLength_min 	:= 15000;
gvl_param.var_productInfo[productID].pocketSumQty		:= 15;
gvl_param.var_productInfo[productID].autoVels.x.vel		:= 300;
gvl_param.var_productInfo[productID].autoVels.x.acc		:= 10000;
gvl_param.var_productInfo[productID].autoVels.x.dcc		:= 10000;
gvl_param.var_productInfo[productID].autoVels.y.vel		:= 150;
gvl_param.var_productInfo[productID].autoVels.y.acc		:= 10000;
gvl_param.var_productInfo[productID].autoVels.y.dcc		:= 10000;
gvl_param.var_productInfo[productID].autoVels.z.vel		:= 150;
gvl_param.var_productInfo[productID].autoVels.z.acc		:= 10000;
gvl_param.var_productInfo[productID].autoVels.z.dcc		:= 10000;
gvl_param.var_productInfo[productID].manaulVels.x.vel	:= 100;
gvl_param.var_productInfo[productID].manaulVels.y.vel	:= 50;
gvl_param.var_productInfo[productID].manaulVels.z.vel	:= 50;

gvl_param.var_productInfo[productID].teachPos.initial.x	:= 950;
gvl_param.var_productInfo[productID].teachPos.initial.y	:= 30;
gvl_param.var_productInfo[productID].teachPos.initial.z	:= 0;
gvl_param.var_productInfo[productID].teachPos.pickUp.x	:= 1250;
gvl_param.var_productInfo[productID].teachPos.pickUp.y	:= 30;
gvl_param.var_productInfo[productID].teachPos.pickUp.z	:= 10;
gvl_param.var_productInfo[productID].teachPos.remove.x	:= 1220;
gvl_param.var_productInfo[productID].teachPos.remove.y	:= 190;
gvl_param.var_productInfo[productID].teachPos.remove.z	:= 10;
//#1
gvl_param.var_productInfo[productID].teachPos.palletize.upperLower[1].cav[1].Pos[1].x := 1007;
gvl_param.var_productInfo[productID].teachPos.palletize.upperLower[1].cav[1].Pos[1].y := 54;
gvl_param.var_productInfo[productID].teachPos.palletize.upperLower[1].cav[1].Pos[1].z := 15;
gvl_param.var_productInfo[productID].teachPos.palletize.upperLower[1].cav[1].Pos[2].x := 1084;
gvl_param.var_productInfo[productID].teachPos.palletize.upperLower[1].cav[1].Pos[2].y := 54;
gvl_param.var_productInfo[productID].teachPos.palletize.upperLower[1].cav[1].Pos[2].z := 15;
gvl_param.var_productInfo[productID].teachPos.palletize.upperLower[1].cav[1].Pos[3].x := 1007;
gvl_param.var_productInfo[productID].teachPos.palletize.upperLower[1].cav[1].Pos[3].y := 256;
gvl_param.var_productInfo[productID].teachPos.palletize.upperLower[1].cav[1].Pos[3].z := 15;
gvl_param.var_productInfo[productID].teachPos.palletize.upperLower[2].cav[1].Pos[1].x := 1007;
gvl_param.var_productInfo[productID].teachPos.palletize.upperLower[2].cav[1].Pos[1].y := 54;
gvl_param.var_productInfo[productID].teachPos.palletize.upperLower[2].cav[1].Pos[1].z := 30;
gvl_param.var_productInfo[productID].teachPos.palletize.upperLower[2].cav[1].Pos[2].x := 1084;
gvl_param.var_productInfo[productID].teachPos.palletize.upperLower[2].cav[1].Pos[2].y := 54;
gvl_param.var_productInfo[productID].teachPos.palletize.upperLower[2].cav[1].Pos[2].z := 30;
gvl_param.var_productInfo[productID].teachPos.palletize.upperLower[2].cav[1].Pos[3].x := 1007;
gvl_param.var_productInfo[productID].teachPos.palletize.upperLower[2].cav[1].Pos[3].y := 256;
gvl_param.var_productInfo[productID].teachPos.palletize.upperLower[2].cav[1].Pos[3].z := 30;
//#2
gvl_param.var_productInfo[productID].teachPos.palletize.upperLower[1].cav[2].Pos[1].x := 886;
gvl_param.var_productInfo[productID].teachPos.palletize.upperLower[1].cav[2].Pos[1].y := 54;
gvl_param.var_productInfo[productID].teachPos.palletize.upperLower[1].cav[2].Pos[1].z := 15;
gvl_param.var_productInfo[productID].teachPos.palletize.upperLower[1].cav[2].Pos[2].x := 963;
gvl_param.var_productInfo[productID].teachPos.palletize.upperLower[1].cav[2].Pos[2].y := 54;
gvl_param.var_productInfo[productID].teachPos.palletize.upperLower[1].cav[2].Pos[2].z := 15;
gvl_param.var_productInfo[productID].teachPos.palletize.upperLower[1].cav[2].Pos[3].x := 886;
gvl_param.var_productInfo[productID].teachPos.palletize.upperLower[1].cav[2].Pos[3].y := 256;
gvl_param.var_productInfo[productID].teachPos.palletize.upperLower[1].cav[2].Pos[3].z := 15;
gvl_param.var_productInfo[productID].teachPos.palletize.upperLower[2].cav[2].Pos[1].x := 886;
gvl_param.var_productInfo[productID].teachPos.palletize.upperLower[2].cav[2].Pos[1].y := 54;
gvl_param.var_productInfo[productID].teachPos.palletize.upperLower[2].cav[2].Pos[1].z := 30;
gvl_param.var_productInfo[productID].teachPos.palletize.upperLower[2].cav[2].Pos[2].x := 963;
gvl_param.var_productInfo[productID].teachPos.palletize.upperLower[2].cav[2].Pos[2].y := 54;
gvl_param.var_productInfo[productID].teachPos.palletize.upperLower[2].cav[2].Pos[2].z := 30;
gvl_param.var_productInfo[productID].teachPos.palletize.upperLower[2].cav[2].Pos[3].x := 886;
gvl_param.var_productInfo[productID].teachPos.palletize.upperLower[2].cav[2].Pos[3].y := 256;
gvl_param.var_productInfo[productID].teachPos.palletize.upperLower[2].cav[2].Pos[3].z := 30;
//#3
gvl_param.var_productInfo[productID].teachPos.palletize.upperLower[1].cav[3].Pos[1].x := 706;
gvl_param.var_productInfo[productID].teachPos.palletize.upperLower[1].cav[3].Pos[1].y := 54;
gvl_param.var_productInfo[productID].teachPos.palletize.upperLower[1].cav[3].Pos[1].z := 15;
gvl_param.var_productInfo[productID].teachPos.palletize.upperLower[1].cav[3].Pos[2].x := 784;
gvl_param.var_productInfo[productID].teachPos.palletize.upperLower[1].cav[3].Pos[2].y := 54;
gvl_param.var_productInfo[productID].teachPos.palletize.upperLower[1].cav[3].Pos[2].z := 15;
gvl_param.var_productInfo[productID].teachPos.palletize.upperLower[1].cav[3].Pos[3].x := 706;
gvl_param.var_productInfo[productID].teachPos.palletize.upperLower[1].cav[3].Pos[3].y := 256;
gvl_param.var_productInfo[productID].teachPos.palletize.upperLower[1].cav[3].Pos[3].z := 15;
gvl_param.var_productInfo[productID].teachPos.palletize.upperLower[2].cav[3].Pos[1].x := 706;
gvl_param.var_productInfo[productID].teachPos.palletize.upperLower[2].cav[3].Pos[1].y := 54;
gvl_param.var_productInfo[productID].teachPos.palletize.upperLower[2].cav[3].Pos[1].z := 30;
gvl_param.var_productInfo[productID].teachPos.palletize.upperLower[2].cav[3].Pos[2].x := 783;
gvl_param.var_productInfo[productID].teachPos.palletize.upperLower[2].cav[3].Pos[2].y := 54;
gvl_param.var_productInfo[productID].teachPos.palletize.upperLower[2].cav[3].Pos[2].z := 30;
gvl_param.var_productInfo[productID].teachPos.palletize.upperLower[2].cav[3].Pos[3].x := 706;
gvl_param.var_productInfo[productID].teachPos.palletize.upperLower[2].cav[3].Pos[3].y := 256;
gvl_param.var_productInfo[productID].teachPos.palletize.upperLower[2].cav[3].Pos[3].z := 30;
//#4
gvl_param.var_productInfo[productID].teachPos.palletize.upperLower[1].cav[4].Pos[1].x := 585;
gvl_param.var_productInfo[productID].teachPos.palletize.upperLower[1].cav[4].Pos[1].y := 54;
gvl_param.var_productInfo[productID].teachPos.palletize.upperLower[1].cav[4].Pos[1].z := 15;
gvl_param.var_productInfo[productID].teachPos.palletize.upperLower[1].cav[4].Pos[2].x := 662;
gvl_param.var_productInfo[productID].teachPos.palletize.upperLower[1].cav[4].Pos[2].y := 54;
gvl_param.var_productInfo[productID].teachPos.palletize.upperLower[1].cav[4].Pos[2].z := 15;
gvl_param.var_productInfo[productID].teachPos.palletize.upperLower[1].cav[4].Pos[3].x := 585;
gvl_param.var_productInfo[productID].teachPos.palletize.upperLower[1].cav[4].Pos[3].y := 256;
gvl_param.var_productInfo[productID].teachPos.palletize.upperLower[1].cav[4].Pos[3].z := 15;
gvl_param.var_productInfo[productID].teachPos.palletize.upperLower[2].cav[4].Pos[1].x := 585;
gvl_param.var_productInfo[productID].teachPos.palletize.upperLower[2].cav[4].Pos[1].y := 54;
gvl_param.var_productInfo[productID].teachPos.palletize.upperLower[2].cav[4].Pos[1].z := 30;
gvl_param.var_productInfo[productID].teachPos.palletize.upperLower[2].cav[4].Pos[2].x := 663;
gvl_param.var_productInfo[productID].teachPos.palletize.upperLower[2].cav[4].Pos[2].y := 54;
gvl_param.var_productInfo[productID].teachPos.palletize.upperLower[2].cav[4].Pos[2].z := 30;
gvl_param.var_productInfo[productID].teachPos.palletize.upperLower[2].cav[4].Pos[3].x := 585;
gvl_param.var_productInfo[productID].teachPos.palletize.upperLower[2].cav[4].Pos[3].y := 256;
gvl_param.var_productInfo[productID].teachPos.palletize.upperLower[2].cav[4].Pos[3].z := 30;
//#5
gvl_param.var_productInfo[productID].teachPos.palletize.upperLower[1].cav[5].Pos[1].x := 406;
gvl_param.var_productInfo[productID].teachPos.palletize.upperLower[1].cav[5].Pos[1].y := 54;
gvl_param.var_productInfo[productID].teachPos.palletize.upperLower[1].cav[5].Pos[1].z := 15;
gvl_param.var_productInfo[productID].teachPos.palletize.upperLower[1].cav[5].Pos[2].x := 484;
gvl_param.var_productInfo[productID].teachPos.palletize.upperLower[1].cav[5].Pos[2].y := 54;
gvl_param.var_productInfo[productID].teachPos.palletize.upperLower[1].cav[5].Pos[2].z := 15;
gvl_param.var_productInfo[productID].teachPos.palletize.upperLower[1].cav[5].Pos[3].x := 406;
gvl_param.var_productInfo[productID].teachPos.palletize.upperLower[1].cav[5].Pos[3].y := 256;
gvl_param.var_productInfo[productID].teachPos.palletize.upperLower[1].cav[5].Pos[3].z := 15;
gvl_param.var_productInfo[productID].teachPos.palletize.upperLower[2].cav[5].Pos[1].x := 405;
gvl_param.var_productInfo[productID].teachPos.palletize.upperLower[2].cav[5].Pos[1].y := 54;
gvl_param.var_productInfo[productID].teachPos.palletize.upperLower[2].cav[5].Pos[1].z := 30;
gvl_param.var_productInfo[productID].teachPos.palletize.upperLower[2].cav[5].Pos[2].x := 483;
gvl_param.var_productInfo[productID].teachPos.palletize.upperLower[2].cav[5].Pos[2].y := 54;
gvl_param.var_productInfo[productID].teachPos.palletize.upperLower[2].cav[5].Pos[2].z := 30;
gvl_param.var_productInfo[productID].teachPos.palletize.upperLower[2].cav[5].Pos[3].x := 405;
gvl_param.var_productInfo[productID].teachPos.palletize.upperLower[2].cav[5].Pos[3].y := 256;
gvl_param.var_productInfo[productID].teachPos.palletize.upperLower[2].cav[5].Pos[3].z := 30;
//#6
gvl_param.var_productInfo[productID].teachPos.palletize.upperLower[1].cav[6].Pos[1].x := 286;
gvl_param.var_productInfo[productID].teachPos.palletize.upperLower[1].cav[6].Pos[1].y := 54;
gvl_param.var_productInfo[productID].teachPos.palletize.upperLower[1].cav[6].Pos[1].z := 15;
gvl_param.var_productInfo[productID].teachPos.palletize.upperLower[1].cav[6].Pos[2].x := 363;
gvl_param.var_productInfo[productID].teachPos.palletize.upperLower[1].cav[6].Pos[2].y := 54;
gvl_param.var_productInfo[productID].teachPos.palletize.upperLower[1].cav[6].Pos[2].z := 15;
gvl_param.var_productInfo[productID].teachPos.palletize.upperLower[1].cav[6].Pos[3].x := 286;
gvl_param.var_productInfo[productID].teachPos.palletize.upperLower[1].cav[6].Pos[3].y := 256;
gvl_param.var_productInfo[productID].teachPos.palletize.upperLower[1].cav[6].Pos[3].z := 15;
gvl_param.var_productInfo[productID].teachPos.palletize.upperLower[2].cav[6].Pos[1].x := 285;
gvl_param.var_productInfo[productID].teachPos.palletize.upperLower[2].cav[6].Pos[1].y := 54;
gvl_param.var_productInfo[productID].teachPos.palletize.upperLower[2].cav[6].Pos[1].z := 30;
gvl_param.var_productInfo[productID].teachPos.palletize.upperLower[2].cav[6].Pos[2].x := 362;
gvl_param.var_productInfo[productID].teachPos.palletize.upperLower[2].cav[6].Pos[2].y := 54;
gvl_param.var_productInfo[productID].teachPos.palletize.upperLower[2].cav[6].Pos[2].z := 30;
gvl_param.var_productInfo[productID].teachPos.palletize.upperLower[2].cav[6].Pos[3].x := 285;
gvl_param.var_productInfo[productID].teachPos.palletize.upperLower[2].cav[6].Pos[3].y := 256;
gvl_param.var_productInfo[productID].teachPos.palletize.upperLower[2].cav[6].Pos[3].z := 30;
//#7
gvl_param.var_productInfo[productID].teachPos.palletize.upperLower[1].cav[7].Pos[1].x := 107;
gvl_param.var_productInfo[productID].teachPos.palletize.upperLower[1].cav[7].Pos[1].y := 54;
gvl_param.var_productInfo[productID].teachPos.palletize.upperLower[1].cav[7].Pos[1].z := 15;
gvl_param.var_productInfo[productID].teachPos.palletize.upperLower[1].cav[7].Pos[2].x := 184;
gvl_param.var_productInfo[productID].teachPos.palletize.upperLower[1].cav[7].Pos[2].y := 54;
gvl_param.var_productInfo[productID].teachPos.palletize.upperLower[1].cav[7].Pos[2].z := 15;
gvl_param.var_productInfo[productID].teachPos.palletize.upperLower[1].cav[7].Pos[3].x := 107;
gvl_param.var_productInfo[productID].teachPos.palletize.upperLower[1].cav[7].Pos[3].y := 256;
gvl_param.var_productInfo[productID].teachPos.palletize.upperLower[1].cav[7].Pos[3].z := 15;
gvl_param.var_productInfo[productID].teachPos.palletize.upperLower[2].cav[7].Pos[1].x := 106;
gvl_param.var_productInfo[productID].teachPos.palletize.upperLower[2].cav[7].Pos[1].y := 54;
gvl_param.var_productInfo[productID].teachPos.palletize.upperLower[2].cav[7].Pos[1].z := 30;
gvl_param.var_productInfo[productID].teachPos.palletize.upperLower[2].cav[7].Pos[2].x := 183;
gvl_param.var_productInfo[productID].teachPos.palletize.upperLower[2].cav[7].Pos[2].y := 54;
gvl_param.var_productInfo[productID].teachPos.palletize.upperLower[2].cav[7].Pos[2].z := 30;
gvl_param.var_productInfo[productID].teachPos.palletize.upperLower[2].cav[7].Pos[3].x := 106;
gvl_param.var_productInfo[productID].teachPos.palletize.upperLower[2].cav[7].Pos[3].y := 256;
gvl_param.var_productInfo[productID].teachPos.palletize.upperLower[2].cav[7].Pos[3].z := 30;
//#8
gvl_param.var_productInfo[productID].teachPos.palletize.upperLower[1].cav[8].Pos[1].x := -13;
gvl_param.var_productInfo[productID].teachPos.palletize.upperLower[1].cav[8].Pos[1].y := 54;
gvl_param.var_productInfo[productID].teachPos.palletize.upperLower[1].cav[8].Pos[1].z := 15;
gvl_param.var_productInfo[productID].teachPos.palletize.upperLower[1].cav[8].Pos[2].x := 63;
gvl_param.var_productInfo[productID].teachPos.palletize.upperLower[1].cav[8].Pos[2].y := 54;
gvl_param.var_productInfo[productID].teachPos.palletize.upperLower[1].cav[8].Pos[2].z := 15;
gvl_param.var_productInfo[productID].teachPos.palletize.upperLower[1].cav[8].Pos[3].x := -13;
gvl_param.var_productInfo[productID].teachPos.palletize.upperLower[1].cav[8].Pos[3].y := 256;
gvl_param.var_productInfo[productID].teachPos.palletize.upperLower[1].cav[8].Pos[3].z := 15;
gvl_param.var_productInfo[productID].teachPos.palletize.upperLower[2].cav[8].Pos[1].x := -14;
gvl_param.var_productInfo[productID].teachPos.palletize.upperLower[2].cav[8].Pos[1].y := 54;
gvl_param.var_productInfo[productID].teachPos.palletize.upperLower[2].cav[8].Pos[1].z := 30;
gvl_param.var_productInfo[productID].teachPos.palletize.upperLower[2].cav[8].Pos[2].x := 62;
gvl_param.var_productInfo[productID].teachPos.palletize.upperLower[2].cav[8].Pos[2].y := 54;
gvl_param.var_productInfo[productID].teachPos.palletize.upperLower[2].cav[8].Pos[2].z := 30;
gvl_param.var_productInfo[productID].teachPos.palletize.upperLower[2].cav[8].Pos[3].x := -14;
gvl_param.var_productInfo[productID].teachPos.palletize.upperLower[2].cav[8].Pos[3].y := 256;
gvl_param.var_productInfo[productID].teachPos.palletize.upperLower[2].cav[8].Pos[3].z := 30;

//sample
gvl_param.var_productInfo[productID].teachPos.sample[1].x := 1263;
gvl_param.var_productInfo[productID].teachPos.sample[1].y := 296;
gvl_param.var_productInfo[productID].teachPos.sample[1].z := 10;
gvl_param.var_productInfo[productID].teachPos.sample[2].x := 1242;
gvl_param.var_productInfo[productID].teachPos.sample[2].y := 296;
gvl_param.var_productInfo[productID].teachPos.sample[2].z := 10;
gvl_param.var_productInfo[productID].teachPos.sample[3].x := 1222;
gvl_param.var_productInfo[productID].teachPos.sample[3].y := 296;
gvl_param.var_productInfo[productID].teachPos.sample[3].z := 10;
gvl_param.var_productInfo[productID].teachPos.sample[4].x := 1202;
gvl_param.var_productInfo[productID].teachPos.sample[4].y := 296;
gvl_param.var_productInfo[productID].teachPos.sample[4].z := 10;
gvl_param.var_productInfo[productID].teachPos.sample[5].x := 1262;
gvl_param.var_productInfo[productID].teachPos.sample[5].y := 187;
gvl_param.var_productInfo[productID].teachPos.sample[5].z := 10;
gvl_param.var_productInfo[productID].teachPos.sample[6].x := 1242;
gvl_param.var_productInfo[productID].teachPos.sample[6].y := 187;
gvl_param.var_productInfo[productID].teachPos.sample[6].z := 10;
gvl_param.var_productInfo[productID].teachPos.sample[7].x := 1222;
gvl_param.var_productInfo[productID].teachPos.sample[7].y := 187;
gvl_param.var_productInfo[productID].teachPos.sample[7].z := 10;
gvl_param.var_productInfo[productID].teachPos.sample[8].x := 1202;
gvl_param.var_productInfo[productID].teachPos.sample[8].y := 187;
gvl_param.var_productInfo[productID].teachPos.sample[8].z := 10;

END_FUNCTION_BLOCK

// ---- FBs/fb_auto.TcPOU
FUNCTION_BLOCK fb_auto
VAR_INPUT
END_VAR
VAR_OUTPUT
END_VAR
VAR
	SFCInit: BOOL;
	trn_paramInitDone: BOOL;
	trn_moveToHomeDone: BOOL;
	trn_removeLensDone: BOOL;
	fbi_paramInit: fb_paramInit;
	var_process: INT;
	flg_tranHomeDone: BOOL;
	flg_sampleHomeDone: BOOL;
	flg_trayHomeDone: BOOL;
	flg_chuckHomeDone: BOOL;
	flg_axisHomeDone: BOOL;
	fbi_lensTranport: fb_lensTranport;
	fbi_palletizeing: fb_palletizeing;
	fbi_gm_measurementModule: fb_gm_measurementModule;
	fbi_gm_transport: fb_gm_transport;
	flg_pushHomeDone: BOOL;
	flg_rotaryHomeDone: BOOL;
	trn_measurementSystemHomeDone: BOOL;
	fbi_debuger : fb_debuger;
	fbi_gateLengthList: fb_gateLengthList;
	fbi_dataSampling: fb_dataSampling;
	timer: TON;
	timer2: TON;
	fbi_gm_removeLens: fb_gm_removeLens;
END_VAR

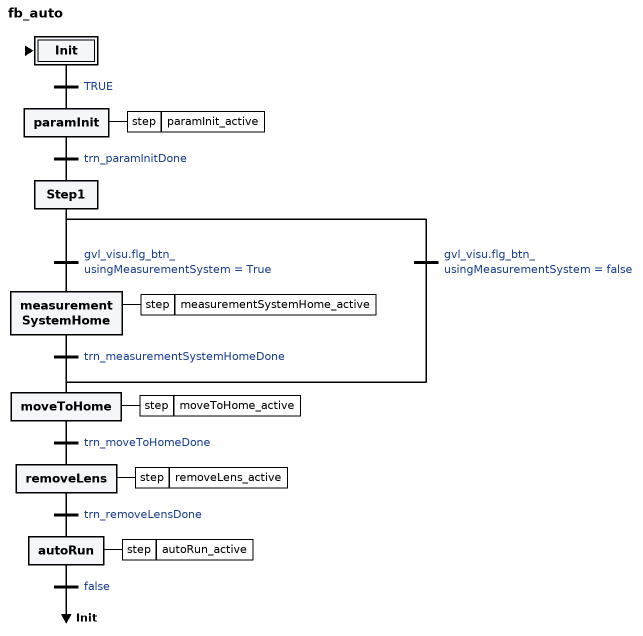
INITIAL_STEP Init:
END_STEP
TRANSITION FROM Init TO paramInit
    := TRUE;
END_TRANSITION
STEP paramInit:
    paramInit_active(N);  // step action
END_STEP
TRANSITION FROM paramInit TO Step1
    := trn_paramInitDone;
END_TRANSITION
STEP Step1:
END_STEP
TRANSITION FROM Step1 TO measurementSystemHome
    := gvl_visu.flg_btn_usingMeasurementSystem = True;
END_TRANSITION
STEP measurementSystemHome:
    measurementSystemHome_active(N);  // step action
END_STEP
TRANSITION FROM measurementSystemHome TO moveToHome
    := trn_measurementSystemHomeDone;
END_TRANSITION
TRANSITION FROM Step1 TO moveToHome
    := gvl_visu.flg_btn_usingMeasurementSystem = false;
END_TRANSITION
STEP moveToHome:
    moveToHome_active(N);  // step action
END_STEP
TRANSITION FROM moveToHome TO removeLens
    := trn_moveToHomeDone;
END_TRANSITION
STEP removeLens:
    removeLens_active(N);  // step action
END_STEP
TRANSITION FROM removeLens TO autoRun
    := trn_removeLensDone;
END_TRANSITION
STEP autoRun:
    autoRun_active(N);  // step action
END_STEP
TRANSITION FROM autoRun TO Init
    := false;
END_TRANSITION

ACTION autoRun_active:
IF autoRun._x AND autoRun.x = FALSE THEN
	THIS^.fbi_lensTranport();
	THIS^.fbi_lensTranport.p_Init := TRUE;
	THIS^.fbi_palletizeing();
	THIS^.fbi_palletizeing.p_Init := TRUE;
	THIS^.fbi_gm_measurementModule.SFCInit := TRUE;
	THIS^.fbi_gm_measurementModule();
	THIS^.fbi_gm_transport();
	THIS^.fbi_gm_transport.p_Init := TRUE;
ELSIF autoRun._x AND autoRun.x THEN
	THIS^.fbi_lensTranport();
	THIS^.fbi_lensTranport.p_Init := FALSE;
	THIS^.fbi_palletizeing();
	THIS^.fbi_palletizeing.p_Init := FALSE;
	IF gvl_visu.flg_btn_usingMeasurementSystem THEN
		THIS^.fbi_gm_measurementModule();
		THIS^.fbi_gm_measurementModule.SFCInit := FALSE;
		THIS^.fbi_gm_transport();
		THIS^.fbi_gm_transport.p_Init := FALSE;
	END_IF
	fbi_dataSampling(
	in_flg_run:= gvl_auto.flg_dataSampling_run, 
	in_var_cavNo:= gvl_auto.buf_cavNo, 
	in_var_pocketNo:= gvl_auto.pocketNo[gvl_auto.buf_cavNo], 
	in_var_gateLength:= gvl_auto.buf_gateLength, 
	in_var_date:= gvl_visu.var_DT, 
	in_flg_nonDefective:= gvl_auto.flg_DataSample_nonDefective, 
	in_flg_defective:= gvl_auto.flg_DataSample_defective, 
	in_flg_sample:= gvl_auto.flg_DataSamle_sample, 
	in_flg_reset:= , 
	ref_dataSet:= gvl_auto.var_DataSet);

	fbi_gateLengthList();
	
	fbi_debuger(
	in_flg_run:= gvl_debug.flg_debug_run, 
	in_flg_start:= gvl_debug.flg_debug_run, 
	in_var_cavQty:= gvl_param.var_productInfo[gvl_param.var_currentProductID].cavQty, 
	out_flg_gateLengthISSuccessed=> gvl_debug.flg_passingMeasurement, 
	out_flg_dummySignal=> , 
	out_flg_lensSetDone=> gvl_debug.out_lensSetDone, 
	out_flg_fiberSens=> gvl_debug.out_fiberSens, 
	out_flg_busy=> gvl_debug.out_busy, 
	out_cav=> gvl_debug.var_cav);
	
END_IF
END_ACTION

ACTION measurementSystemHome_active:
IF measurementSystemHome._x AND measurementSystemHome.x = FALSE THEN
	trn_measurementSystemHomeDone := FALSE;
	gvl_auto.gm_rotaryPowerOn := FALSE;
	var_process := 0;
ELSIF measurementSystemHome._x AND measurementSystemHome.x THEN
	IF gvl_visu.flg_btn_usingMeasurementSystem THEN
		CASE var_process OF
			0://insert parameter
				gvl_solv.fbi_gm_ejector.in_flg_run := FALSE;
				gvl_solv.fbi_gm_chuck.in_flg_run := FALSE;
				gvl_solv.fbi_gm_push.in_flg_run := FALSE;
				gvl_solv.fbi_gm_pickup.in_flg_run := FALSE;
				gvl_solv.fbi_gm_rotary.in_flg_run := FALSE;
				gvl_solv.fbi_gm_stamp.in_flg_run := FALSE;
				gvl_elecylinder.fbi_gm_axisPickUp.in_flg_run := FALSE;
				gvl_elecylinder.fbi_gm_axisTransport.in_flg_run := FALSE;
				gvl_solv.fbi_gm_ejector.in_var_vacMode := eP_ejeVacMode.halt;
				gvl_solv.fbi_gm_chuck.in_var_moveMode := eP_svMoveMode.svA;
				gvl_solv.fbi_gm_push.in_var_moveMode := eP_svMoveMode.svA;
				gvl_solv.fbi_gm_pickup.in_var_moveMode := eP_svMoveMode.svA;
				gvl_solv.fbi_gm_rotary.in_var_moveMode := eP_svMoveMode.svA;
				gvl_solv.fbi_gm_stamp.in_var_moveMode := eP_svMoveMode.svA;
				gvl_elecylinder.fbi_gm_axisPickUp.in_var_moveMode := eP_eleMoveMode.eleA;
				gvl_elecylinder.fbi_gm_axisTransport.in_var_moveMode := eP_eleMoveMode.eleA;
				gvl_axis.ref_r.Position := gvl_param.var_productInfo[gvl_param.var_currentProductID].teachPos.gm_rotary.origin;
				gvl_auto.gm_rotaryPowerOn := TRUE;
				IF gvl_axis.fbi_mc_powerR.Status THEN
					var_process := 1;
				END_IF
			1://first move
				gvl_solv.fbi_gm_ejector.in_flg_run := TRUE;
				gvl_solv.fbi_gm_chuck.in_flg_run := TRUE;
				gvl_solv.fbi_gm_push.in_flg_run := TRUE;
				gvl_elecylinder.fbi_gm_axisPickUp.in_flg_run := TRUE;
				gvl_elecylinder.fbi_gm_axisTransport.in_flg_run := TRUE;
				IF gvl_solv.ref_gm_chuck.in.in_flg_sensA AND
				   gvl_solv.ref_gm_push.in.in_flg_sensA AND
				   gvl_elecylinder.ref_gm_axisPickUp.input.in_flg_sensA AND 
				   gvl_elecylinder.ref_gm_axisTransport.input.in_flg_sensA THEN
				   	gvl_solv.fbi_gm_ejector.in_flg_run := FALSE;
					gvl_solv.fbi_gm_chuck.in_flg_run := FALSE;
					gvl_solv.fbi_gm_push.in_flg_run := FALSE;
					gvl_elecylinder.fbi_gm_axisPickUp .in_flg_run := FALSE;
					gvl_elecylinder.fbi_gm_axisTransport.in_flg_run := FALSE;
					var_process := 2;
				END_IF
			2://second move	
				gvl_axis.ref_r.Execute := TRUE;
				IF gvl_axis.ref_r.Done THEN
					gvl_axis.ref_r.Execute := FALSE;
					var_process := 3;
				END_IF
			3://third move
				gvl_solv.fbi_gm_pickup.in_flg_run := TRUE;
				gvl_solv.fbi_gm_rotary.in_flg_run := TRUE;
				gvl_solv.fbi_gm_stamp.in_flg_run := TRUE;
				IF gvl_solv.ref_gm_pickUp.in.in_flg_sensA AND gvl_solv.ref_gm_rotary.in.in_flg_sensA AND gvl_solv.ref_gm_stamp.in.in_flg_sensA THEN
					var_process := 4;
				END_IF
			4:	
				trn_measurementSystemHomeDone := TRUE;
		END_CASE
		IF gvl_axis.ref_r.Error THEN
			gvl_axis.ref_r.Execute := false;
			var_process := 100;
		END_IF
	ELSE
		trn_measurementSystemHomeDone := TRUE;
	END_IF
END_IF
END_ACTION

ACTION moveToHome_active:
IF moveToHome._x AND moveToHome.x = FALSE THEN
	var_process := 0;
	trn_moveToHomeDone := FALSE;
	gvl_auto.motorPowerOn := FALSE;
ELSIF moveToHome._x AND moveToHome.x THEN
	CASE var_process OF
		0:
			gvl_auto.motorPowerOn := TRUE;
			IF gvl_axis.flg_motorReady THEN
				var_process := 1;
			END_IF
		1://move axisZ
			gvl_axis.ref_z.Position := 0;
			gvl_axis.ref_z.Execute := TRUE;
			IF gvl_axis.ref_z.Done THEN
				gvl_axis.ref_z.Execute := FALSE;
				var_process := 2;
			END_IF
		2://insert parameter
			gvl_solv.fbi_push.in_flg_run := FALSE;
			gvl_elecylinder.fbi_axisTransport.in_var_moveMode := eP_eleMoveMode.eleA;
			gvl_elecylinder.fbi_axisSample.in_var_moveMode := eP_eleMoveMode.eleA;
			gvl_elecylinder.fbi_axisRotary.in_var_moveMode := eP_eleMoveMode.eleA;
			gvl_solv.fbi_chuck.in_var_moveMode := eP_svMoveMode.svA;
			gvl_solv.fbi_push.in_var_moveMode := eP_svMoveMode.svA;
			gvl_elecylinder.fbi_axisTransport.in_flg_run := FALSE;
			gvl_elecylinder.fbi_axisSample.in_flg_run := FALSE;
			gvl_elecylinder.fbi_axisRotary.in_flg_run := FALSE;
			gvl_solv.fbi_chuck.in_flg_run := FALSE;
			gvl_solv.fbi_push.in_flg_run := FALSE;
			gvl_axis.fbi_motionControler.in_flg_start := false;
			gvl_axis.fbi_motionControler.in_var_targetPosX := gvl_param.var_productInfo[gvl_param.var_currentProductID].teachPos.initial.x;
			gvl_axis.fbi_motionControler.in_var_targetPosY := gvl_param.var_productInfo[gvl_param.var_currentProductID].teachPos.initial.y;
			gvl_axis.fbi_motionControler.in_var_targetPosZ := gvl_param.var_productInfo[gvl_param.var_currentProductID].teachPos.initial.z;
			gvl_axis.fbi_motionControler.in_var_direction := eP_motionDirection.XYZ;
			var_process := 3;
		3://moving start
			gvl_elecylinder.fbi_axisTransport.in_flg_run := TRUE;
			gvl_elecylinder.fbi_axisSample.in_flg_run := TRUE;
			gvl_elecylinder.fbi_axisRotary.in_flg_run := TRUE;
			gvl_solv.fbi_chuck.in_flg_run := TRUE;
			gvl_solv.fbi_push.in_flg_run := TRUE;
			gvl_axis.fbi_motionControler.in_flg_start := TRUE;
			IF gvl_elecylinder.fbi_axisTransport.out_flg_Done THEN
				flg_tranHomeDone := TRUE;
			END_IF
			IF gvl_elecylinder.fbi_axisSample.out_flg_Done THEN
				flg_sampleHomeDone := TRUE;
			END_IF
			IF gvl_elecylinder.fbi_axisRotary.out_flg_Done THEN
				flg_rotaryHomeDone := TRUE;
			END_IF
			IF gvl_solv.fbi_chuck.out_flg_Done THEN
				flg_chuckHomeDone := TRUE;
			END_IF
			IF gvl_solv.fbi_push.out_flg_Done THEN
				flg_pushHomeDone := TRUE;
			END_IF
			IF gvl_axis.fbi_motionControler.out_flg_Done THEN
				flg_axisHomeDone := TRUE;
			END_IF 
			IF flg_tranHomeDone AND flg_sampleHomeDone AND flg_chuckHomeDone AND flg_axisHomeDone AND flg_pushHomeDone AND flg_rotaryHomeDone THEN
				var_process := 4;
			END_IF
		4://clear flag
			flg_tranHomeDone := FALSE;
			flg_sampleHomeDone := FALSE;
			flg_chuckHomeDone := FALSE;
			flg_pushHomeDone := FALSE;
			flg_axisHomeDone := FALSE;
			flg_rotaryHomeDone := FALSE;
			gvl_elecylinder.fbi_axisTransport.in_flg_run := FALSE;
			gvl_elecylinder.fbi_axisSample.in_flg_run := FALSE;
			gvl_elecylinder.fbi_axisTrayChange.in_flg_run := FALSE;
			gvl_elecylinder.fbi_axisRotary.in_flg_run := FALSE;
			gvl_solv.fbi_chuck.in_flg_run := FALSE;
			gvl_solv.fbi_push.in_flg_run := FALSE;
			gvl_axis.fbi_motionControler.in_flg_start := FALSE;
			var_process := 5;
		5://check position
			trn_moveToHomeDone := TRUE;			
	END_CASE
END_IF
END_ACTION

PROPERTY p_Init : BOOL
GET
p_Init := THIS^.SFCInit;
END_GET
SET
THIS^.SFCInit := p_Init;
END_SET
END_PROPERTY

ACTION paramInit_active:
IF paramInit._x AND paramInit.x = FALSE THEN
	trn_paramInitDone := FALSE;
	fbi_paramInit.in_flg_run := FALSE;
	THIS^.fbi_lensTranport.p_Init := TRUE;
	THIS^.fbi_lensTranport();
	THIS^.fbi_palletizeing.p_Init := TRUE;
	THIS^.fbi_palletizeing();
	THIS^.fbi_gm_measurementModule.SFCInit := TRUE;
	THIS^.fbi_gm_measurementModule();
	THIS^.fbi_gm_transport();
	THIS^.fbi_gm_transport.p_Init := TRUE;
ELSIF paramInit._x AND paramInit.x THEN
	gvl_auto.gateLengthIsPassed := FALSE;
	gvl_auto.pickUpLnesDone := FALSE;
	gvl_auto.lensVacuumDone := FALSE;
	gvl_auto.requirementToPickUpLens := FALSE;
	gvl_gm.flg_requestPickup := FALSE;
	gvl_gm.flg_lensSetDoneFromGM := FALSE;
	gvl_gm.flg_lensRequest := FALSE;
	gvl_gm.flg_lensPickUpDone := FALSE;
	gvl_debug.flg_debug_run := FALSE;
	gvl_debug.flg_stampDone :=FALSE;
	gvl_debug.flg_stampReady := FALSE;
	gvl_debug.flg_check_quality:= FALSE;
	gvl_debug.flg_to_measurement:= FALSE;
	gvl_debug.flg_to_stocker:= FALSE;
	gvl_visu.flg_btn_vacSensOn := FALSE;
	gvl_visu.flg_btn_gm_motorPower := FALSE;
	gvl_visu.flg_btn_buzzer_silent := FALSE;
	gvl_visu.flg_powerOn := FALSE;
	fbi_paramInit.in_flg_run := TRUE;
	IF fbi_paramInit.out_flg_done THEN
		fbi_paramInit.in_flg_run := FALSE;
		trn_paramInitDone := TRUE;
	END_IF
END_IF

fbi_paramInit(in_flg_run:= , out_flg_done=> );
END_ACTION

